REGION Network 7: 380A1 FB
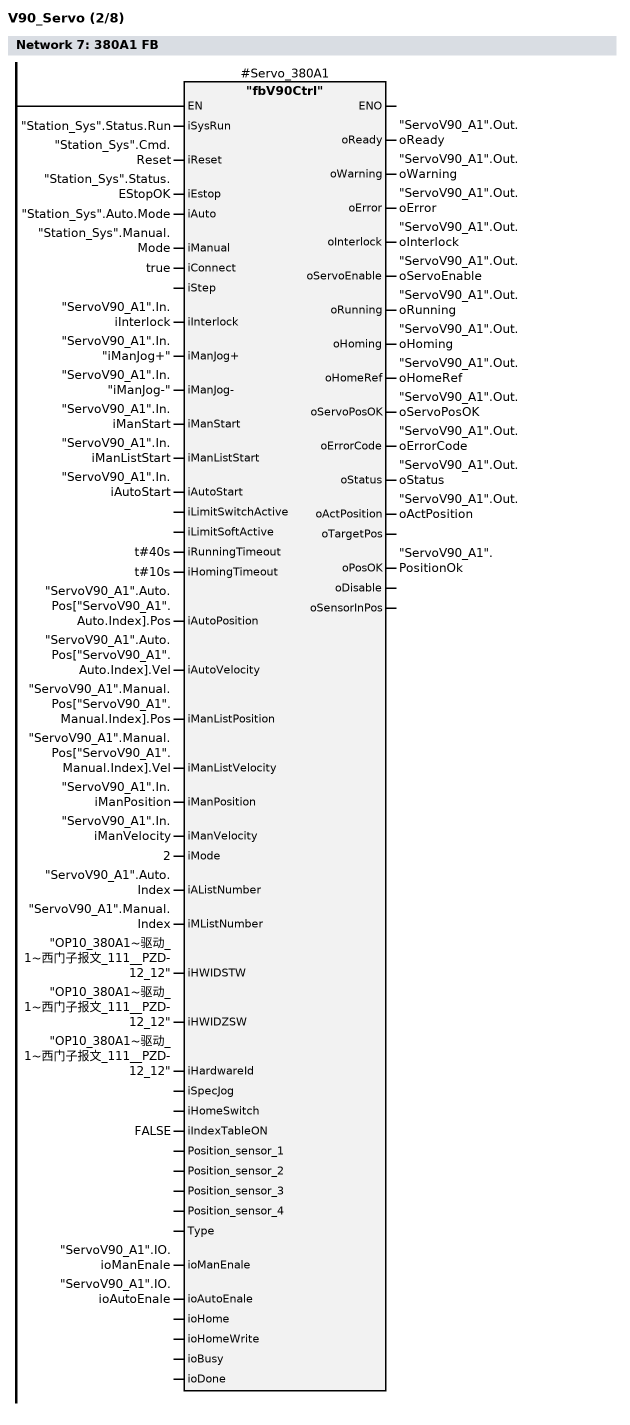
   RUNG wire#powerrail
      #Servo_380A1(iSysRun := "Station_Sys".Status.Run, iReset := "Station_Sys".Cmd.Reset, iEstop := "Station_Sys".Status.EStopOK, iAuto := "Station_Sys".Auto.Mode, iManual := "Station_Sys".Manual.Mode, iConnect := true, iStep :=, iInterlock := "ServoV90_A1".In.iInterlock, "iManJog+" := "ServoV90_A1".In."iManJog+", "iManJog-" := "ServoV90_A1".In."iManJog-", iManStart := "ServoV90_A1".In.iManStart, iManListStart := "ServoV90_A1".In.iManListStart, iAutoStart := "ServoV90_A1".In.iAutoStart, iLimitSwitchActive :=, iLimitSoftActive :=, iRunningTimeout := t#40s, iHomingTimeout := t#10s, iAutoPosition := "ServoV90_A1".Auto.Pos["ServoV90_A1".Auto.Index].Pos, iAutoVelocity := "ServoV90_A1".Auto.Pos["ServoV90_A1".Auto.Index].Vel, iManListPosition := "ServoV90_A1".Manual.Pos["ServoV90_A1".Manual.Index].Pos, iManListVelocity := "ServoV90_A1".Manual.Pos["ServoV90_A1".Manual.Index].Vel, iManPosition := "ServoV90_A1".In.iManPosition, iManVelocity := "ServoV90_A1".In.iManVelocity, iMode := 2, iAListNumber := "ServoV90_A1".Auto.Index, iMListNumber := "ServoV90_A1".Manual.Index, iHWIDSTW := "OP10_380A1~驱动_1~西门子报文_111__PZD-12_12", iHWIDZSW := "OP10_380A1~驱动_1~西门子报文_111__PZD-12_12", iHardwareId := "OP10_380A1~驱动_1~西门子报文_111__PZD-12_12", iSpecJog :=, iHomeSwitch :=, iIndexTableON := FALSE, Position_sensor_1 :=, Position_sensor_2 :=, Position_sensor_3 :=, Position_sensor_4 :=, "Type" :=, ioManEnale := "ServoV90_A1".IO.ioManEnale, ioAutoEnale := "ServoV90_A1".IO.ioAutoEnale, ioHome :=, ioHomeWrite :=, ioBusy :=, ioDone :=, oReady => "ServoV90_A1".Out.oReady, oWarning => "ServoV90_A1".Out.oWarning, oError => "ServoV90_A1".Out.oError, oInterlock => "ServoV90_A1".Out.oInterlock, oServoEnable => "ServoV90_A1".Out.oServoEnable, oRunning => "ServoV90_A1".Out.oRunning, oHoming => "ServoV90_A1".Out.oHoming, oHomeRef => "ServoV90_A1".Out.oHomeRef, oServoPosOK => "ServoV90_A1".Out.oServoPosOK, oErrorCode => "ServoV90_A1".Out.oErrorCode, oStatus => "ServoV90_A1".Out.oStatus, oActPosition => "ServoV90_A1".Out.oActPosition, oTargetPos =>, oPosOK => "ServoV90_A1".PositionOk, oDisable =>, oSensorInPos =>)
   END_RUNG
   // the same network as SCL:
   #Servo_380A1(iSysRun := "Station_Sys".Status.Run,   // "fbV90Ctrl"
                iReset := "Station_Sys".Cmd.Reset,
                iEstop := "Station_Sys".Status.EStopOK,
                iAuto := "Station_Sys".Auto.Mode,
                iManual := "Station_Sys".Manual.Mode,
                iConnect := true,
                iInterlock := "ServoV90_A1".In.iInterlock,
                "iManJog+" := "ServoV90_A1".In."iManJog+",
                "iManJog-" := "ServoV90_A1".In."iManJog-",
                iManStart := "ServoV90_A1".In.iManStart,
                iManListStart := "ServoV90_A1".In.iManListStart,
                iAutoStart := "ServoV90_A1".In.iAutoStart,
                iRunningTimeout := t#40s,
                iHomingTimeout := t#10s,
                iAutoPosition := "ServoV90_A1".Auto.Pos["ServoV90_A1".Auto.Index].Pos,
                iAutoVelocity := "ServoV90_A1".Auto.Pos["ServoV90_A1".Auto.Index].Vel,
                iManListPosition := "ServoV90_A1".Manual.Pos["ServoV90_A1".Manual.Index].Pos,
                iManListVelocity := "ServoV90_A1".Manual.Pos["ServoV90_A1".Manual.Index].Vel,
                iManPosition := "ServoV90_A1".In.iManPosition,
                iManVelocity := "ServoV90_A1".In.iManVelocity,
                iMode := 2,
                iAListNumber := "ServoV90_A1".Auto.Index,
                iMListNumber := "ServoV90_A1".Manual.Index,
                iHWIDSTW := "OP10_380A1~驱动_1~西门子报文_111__PZD-12_12",
                iHWIDZSW := "OP10_380A1~驱动_1~西门子报文_111__PZD-12_12",
                iHardwareId := "OP10_380A1~驱动_1~西门子报文_111__PZD-12_12",
                iIndexTableON := FALSE,
                ioManEnale := "ServoV90_A1".IO.ioManEnale,
                ioAutoEnale := "ServoV90_A1".IO.ioAutoEnale,
                oReady => "ServoV90_A1".Out.oReady,
                oWarning => "ServoV90_A1".Out.oWarning,
                oError => "ServoV90_A1".Out.oError,
                oInterlock => "ServoV90_A1".Out.oInterlock,
                oServoEnable => "ServoV90_A1".Out.oServoEnable,
                oRunning => "ServoV90_A1".Out.oRunning,
                oHoming => "ServoV90_A1".Out.oHoming,
                oHomeRef => "ServoV90_A1".Out.oHomeRef,
                oServoPosOK => "ServoV90_A1".Out.oServoPosOK,
                oErrorCode => "ServoV90_A1".Out.oErrorCode,
                oStatus => "ServoV90_A1".Out.oStatus,
                oActPosition => "ServoV90_A1".Out.oActPosition,
                oPosOK => "ServoV90_A1".PositionOk);
END_REGION

REGION Network 8 (SCL): 故障显示 / Fault indication
   //"ST70_DeviceError".Servo1.ServoDriverError := "ServoV90_A1".Out.oError;
END_REGION

REGION Network 9: <<<<<<<<<<<<<<<<<<<<<381A1 Servo>>>>>>>>>>>>>>>>>>>>>>>>>
END_REGION

REGION Network 10: negtive motion/action/...automaticly
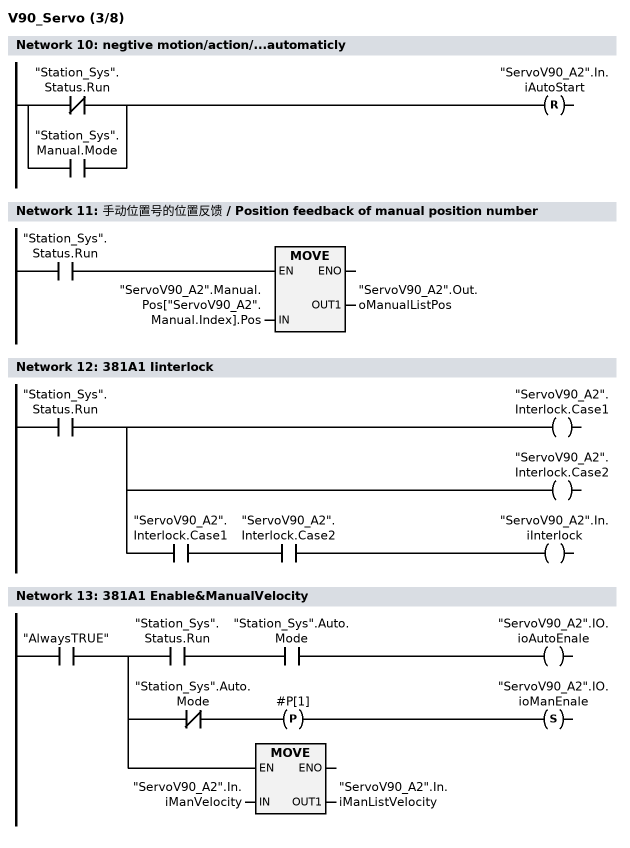
   RUNG wire#powerrail
      I_Contact( "Station_Sys".Status.Run )
      wire#w1
      R_Coil( "ServoV90_A2".In.iAutoStart )
   END_RUNG
   RUNG wire#powerrail
      Contact( "Station_Sys".Manual.Mode )
   END_RUNG wire#w1
   // the same network as SCL:
   IF NOT "Station_Sys".Status.Run OR "Station_Sys".Manual.Mode THEN
       "ServoV90_A2".In.iAutoStart := FALSE;
   END_IF;
END_REGION

REGION Network 11: 手动位置号的位置反馈 / Position feedback of manual position number
   RUNG wire#powerrail
      Contact( "Station_Sys".Status.Run )
      Move(in := "ServoV90_A2".Manual.Pos["ServoV90_A2".Manual.Index].Pos, out1 => "ServoV90_A2".Out.oManualListPos)
   END_RUNG
   // the same network as SCL:
   IF "Station_Sys".Status.Run THEN
       "ServoV90_A2".Out.oManualListPos := "ServoV90_A2".Manual.Pos["ServoV90_A2".Manual.Index].Pos;
   END_IF;
END_REGION

REGION Network 12: 381A1 Iinterlock
   RUNG wire#powerrail
      Contact( "Station_Sys".Status.Run )
      wire#w1
      Coil( "ServoV90_A2".Interlock.Case1 )
   END_RUNG
   RUNG wire#w1
      Coil( "ServoV90_A2".Interlock.Case2 )
   END_RUNG
   RUNG wire#w1
      Contact( "ServoV90_A2".Interlock.Case1 )
      Contact( "ServoV90_A2".Interlock.Case2 )
      Coil( "ServoV90_A2".In.iInterlock )
   END_RUNG
   // the same network as SCL:
   "ServoV90_A2".Interlock.Case1 := "Station_Sys".Status.Run;
   "ServoV90_A2".Interlock.Case2 := "Station_Sys".Status.Run;
   "ServoV90_A2".In.iInterlock := "Station_Sys".Status.Run AND "ServoV90_A2".Interlock.Case1 AND "ServoV90_A2".Interlock.Case2;
END_REGION

REGION Network 13: 381A1 Enable&ManualVelocity
   RUNG wire#powerrail
      Contact( "AlwaysTRUE" )
      wire#w1
      Contact( "Station_Sys".Status.Run )
      Contact( "Station_Sys".Auto.Mode )
      Coil( "ServoV90_A2".IO.ioAutoEnale )
   END_RUNG
   RUNG wire#w1
      I_Contact( "Station_Sys".Auto.Mode )
      P_Trig( #P[1] )
      S_Coil( "ServoV90_A2".IO.ioManEnale )
   END_RUNG
   RUNG wire#w1
      Move(in := "ServoV90_A2".In.iManVelocity, out1 => "ServoV90_A2".In.iManListVelocity)
   END_RUNG
   // the same network as SCL:
   "ServoV90_A2".IO.ioAutoEnale := "AlwaysTRUE" AND "Station_Sys".Status.Run AND "Station_Sys".Auto.Mode;
   #_w1 := "AlwaysTRUE" AND NOT "Station_Sys".Auto.Mode;
   #_w2 := #_w1 AND NOT #P[1];   // rising edge
   #P[1] := #_w1;
   IF #_w2 THEN "ServoV90_A2".IO.ioManEnale := TRUE; END_IF;
   IF "AlwaysTRUE" THEN "ServoV90_A2".In.iManListVelocity := "ServoV90_A2".In.iManVelocity; END_IF;
END_REGION

REGION Network 14 (SCL): 381A1 RecipePosition
    IF "Station_Sys".Status.Run THEN
        "ServoV90_A2".Manual.Pos[1].Pos := "ServoV90_A2".Auto.Pos[1].Pos := REAL_TO_DINT("Parameter".AxisRun.Axis[2].Pos1.Position*1000);
       "ServoV90_A2".Manual.Pos[1].Vel := "ServoV90_A2".Auto.Pos[1].Vel := "Parameter".AxisRun.Axis[2].Pos1.Speed;

       "ServoV90_A2".Manual.Pos[2].Pos := "ServoV90_A2".Auto.Pos[2].Pos := REAL_TO_DINT("Parameter".AxisRun.Axis[2].Pos2.Position*1000);
       "ServoV90_A2".Manual.Pos[2].Vel := "ServoV90_A2".Auto.Pos[2].Vel := "Parameter".AxisRun.Axis[2].Pos2.Speed;

       "ServoV90_A2".Manual.Pos[3].Pos := "ServoV90_A2".Auto.Pos[3].Pos := REAL_TO_DINT("Parameter".AxisRun.Axis[2].Pos3.Position*1000);
       "ServoV90_A2".Manual.Pos[3].Vel := "ServoV90_A2".Auto.Pos[3].Vel := "Parameter".AxisRun.Axis[2].Pos3.Speed;

       "ServoV90_A2".Manual.Pos[4].Pos := "ServoV90_A2".Auto.Pos[4].Pos := REAL_TO_DINT("Parameter".AxisRun.Axis[2].Pos4.Position*1000);
       "ServoV90_A2".Manual.Pos[4].Vel := "ServoV90_A2".Auto.Pos[4].Vel := "Parameter".AxisRun.Axis[2].Pos4.Speed;

       "ServoV90_A2".Manual.Pos[5].Pos := "ServoV90_A2".Auto.Pos[5].Pos := REAL_TO_DINT("Parameter".AxisRun.Axis[2].Pos5.Position*1000);
       "ServoV90_A2".Manual.Pos[5].Vel := "ServoV90_A2".Auto.Pos[5].Vel := "Parameter".AxisRun.Axis[2].Pos5.Speed;

       "ServoV90_A2".Manual.Pos[6].Pos := "ServoV90_A2".Auto.Pos[6].Pos := REAL_TO_DINT("Parameter".AxisRun.Axis[2].Pos6.Position*1000);
       "ServoV90_A2".Manual.Pos[6].Vel := "ServoV90_A2".Auto.Pos[6].Vel := "Parameter".AxisRun.Axis[2].Pos6.Speed;

       "ServoV90_A2".Manual.Pos[7].Pos := "ServoV90_A2".Auto.Pos[7].Pos := REAL_TO_DINT("Parameter".AxisRun.Axis[2].Pos7.Position*1000);
       "ServoV90_A2".Manual.Pos[7].Vel := "ServoV90_A2".Auto.Pos[7].Vel := "Parameter".AxisRun.Axis[2].Pos7.Speed;

       "ServoV90_A2".Manual.Pos[8].Pos := "ServoV90_A2".Auto.Pos[8].Pos := REAL_TO_DINT("Parameter".AxisRun.Axis[2].Pos8.Position*1000);
       "ServoV90_A2".Manual.Pos[8].Vel := "ServoV90_A2".Auto.Pos[8].Vel := "Parameter".AxisRun.Axis[2].Pos8.Speed;

       "ServoV90_A2".Manual.Pos[9].Pos := "ServoV90_A2".Auto.Pos[9].Pos := REAL_TO_DINT("Parameter".AxisRun.Axis[2].Pos9.Position*1000);
       "ServoV90_A2".Manual.Pos[9].Vel := "ServoV90_A2".Auto.Pos[9].Vel := "Parameter".AxisRun.Axis[2].Pos9.Speed;

       "ServoV90_A2".Manual.Pos[10].Pos := "ServoV90_A2".Auto.Pos[10].Pos := REAL_TO_DINT("Parameter".AxisRun.Axis[2].Pos10.Position*1000);
       "ServoV90_A2".Manual.Pos[10].Vel := "ServoV90_A2".Auto.Pos[10].Vel := "Parameter".AxisRun.Axis[2].Pos10.Speed;
   END_IF;
END_REGION

REGION Network 15: 381A1 FB
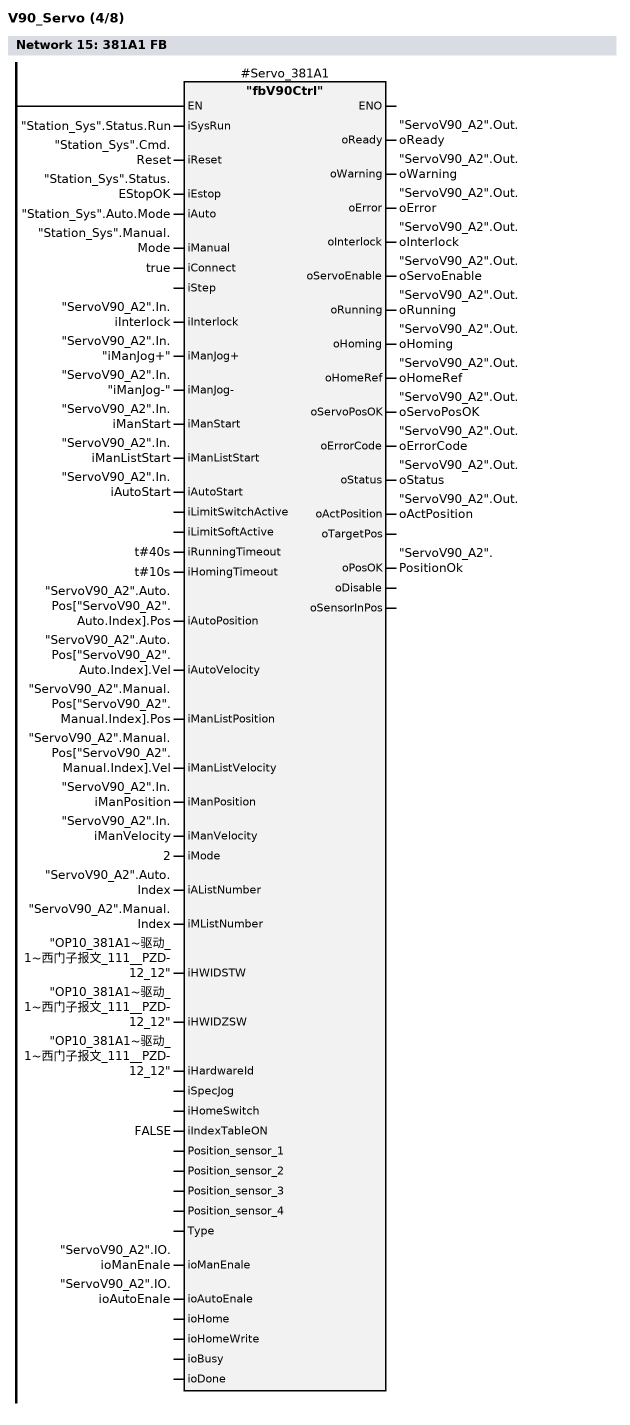
   RUNG wire#powerrail
      #Servo_381A1(iSysRun := "Station_Sys".Status.Run, iReset := "Station_Sys".Cmd.Reset, iEstop := "Station_Sys".Status.EStopOK, iAuto := "Station_Sys".Auto.Mode, iManual := "Station_Sys".Manual.Mode, iConnect := true, iStep :=, iInterlock := "ServoV90_A2".In.iInterlock, "iManJog+" := "ServoV90_A2".In."iManJog+", "iManJog-" := "ServoV90_A2".In."iManJog-", iManStart := "ServoV90_A2".In.iManStart, iManListStart := "ServoV90_A2".In.iManListStart, iAutoStart := "ServoV90_A2".In.iAutoStart, iLimitSwitchActive :=, iLimitSoftActive :=, iRunningTimeout := t#40s, iHomingTimeout := t#10s, iAutoPosition := "ServoV90_A2".Auto.Pos["ServoV90_A2".Auto.Index].Pos, iAutoVelocity := "ServoV90_A2".Auto.Pos["ServoV90_A2".Auto.Index].Vel, iManListPosition := "ServoV90_A2".Manual.Pos["ServoV90_A2".Manual.Index].Pos, iManListVelocity := "ServoV90_A2".Manual.Pos["ServoV90_A2".Manual.Index].Vel, iManPosition := "ServoV90_A2".In.iManPosition, iManVelocity := "ServoV90_A2".In.iManVelocity, iMode := 2, iAListNumber := "ServoV90_A2".Auto.Index, iMListNumber := "ServoV90_A2".Manual.Index, iHWIDSTW := "OP10_381A1~驱动_1~西门子报文_111__PZD-12_12", iHWIDZSW := "OP10_381A1~驱动_1~西门子报文_111__PZD-12_12", iHardwareId := "OP10_381A1~驱动_1~西门子报文_111__PZD-12_12", iSpecJog :=, iHomeSwitch :=, iIndexTableON := FALSE, Position_sensor_1 :=, Position_sensor_2 :=, Position_sensor_3 :=, Position_sensor_4 :=, "Type" :=, ioManEnale := "ServoV90_A2".IO.ioManEnale, ioAutoEnale := "ServoV90_A2".IO.ioAutoEnale, ioHome :=, ioHomeWrite :=, ioBusy :=, ioDone :=, oReady => "ServoV90_A2".Out.oReady, oWarning => "ServoV90_A2".Out.oWarning, oError => "ServoV90_A2".Out.oError, oInterlock => "ServoV90_A2".Out.oInterlock, oServoEnable => "ServoV90_A2".Out.oServoEnable, oRunning => "ServoV90_A2".Out.oRunning, oHoming => "ServoV90_A2".Out.oHoming, oHomeRef => "ServoV90_A2".Out.oHomeRef, oServoPosOK => "ServoV90_A2".Out.oServoPosOK, oErrorCode => "ServoV90_A2".Out.oErrorCode, oStatus => "ServoV90_A2".Out.oStatus, oActPosition => "ServoV90_A2".Out.oActPosition, oTargetPos =>, oPosOK => "ServoV90_A2".PositionOk, oDisable =>, oSensorInPos =>)
   END_RUNG
   // the same network as SCL:
   #Servo_381A1(iSysRun := "Station_Sys".Status.Run,   // "fbV90Ctrl"
                iReset := "Station_Sys".Cmd.Reset,
                iEstop := "Station_Sys".Status.EStopOK,
                iAuto := "Station_Sys".Auto.Mode,
                iManual := "Station_Sys".Manual.Mode,
                iConnect := true,
                iInterlock := "ServoV90_A2".In.iInterlock,
                "iManJog+" := "ServoV90_A2".In."iManJog+",
                "iManJog-" := "ServoV90_A2".In."iManJog-",
                iManStart := "ServoV90_A2".In.iManStart,
                iManListStart := "ServoV90_A2".In.iManListStart,
                iAutoStart := "ServoV90_A2".In.iAutoStart,
                iRunningTimeout := t#40s,
                iHomingTimeout := t#10s,
                iAutoPosition := "ServoV90_A2".Auto.Pos["ServoV90_A2".Auto.Index].Pos,
                iAutoVelocity := "ServoV90_A2".Auto.Pos["ServoV90_A2".Auto.Index].Vel,
                iManListPosition := "ServoV90_A2".Manual.Pos["ServoV90_A2".Manual.Index].Pos,
                iManListVelocity := "ServoV90_A2".Manual.Pos["ServoV90_A2".Manual.Index].Vel,
                iManPosition := "ServoV90_A2".In.iManPosition,
                iManVelocity := "ServoV90_A2".In.iManVelocity,
                iMode := 2,
                iAListNumber := "ServoV90_A2".Auto.Index,
                iMListNumber := "ServoV90_A2".Manual.Index,
                iHWIDSTW := "OP10_381A1~驱动_1~西门子报文_111__PZD-12_12",
                iHWIDZSW := "OP10_381A1~驱动_1~西门子报文_111__PZD-12_12",
                iHardwareId := "OP10_381A1~驱动_1~西门子报文_111__PZD-12_12",
                iIndexTableON := FALSE,
                ioManEnale := "ServoV90_A2".IO.ioManEnale,
                ioAutoEnale := "ServoV90_A2".IO.ioAutoEnale,
                oReady => "ServoV90_A2".Out.oReady,
                oWarning => "ServoV90_A2".Out.oWarning,
                oError => "ServoV90_A2".Out.oError,
                oInterlock => "ServoV90_A2".Out.oInterlock,
                oServoEnable => "ServoV90_A2".Out.oServoEnable,
                oRunning => "ServoV90_A2".Out.oRunning,
                oHoming => "ServoV90_A2".Out.oHoming,
                oHomeRef => "ServoV90_A2".Out.oHomeRef,
                oServoPosOK => "ServoV90_A2".Out.oServoPosOK,
                oErrorCode => "ServoV90_A2".Out.oErrorCode,
                oStatus => "ServoV90_A2".Out.oStatus,
                oActPosition => "ServoV90_A2".Out.oActPosition,
                oPosOK => "ServoV90_A2".PositionOk);
END_REGION

REGION Network 16 (SCL): 故障显示 / Fault indication
   //"ST70_DeviceError".Servo2.ServoDriverError := "ServoV90_A2".Out.oError;
END_REGION

REGION Network 17: <<<<<<<<<<<<<<<<<<<<<382A1 Servo>>>>>>>>>>>>>>>>>>>>>>>>>
END_REGION

REGION Network 18: negtive motion/action/...automaticly
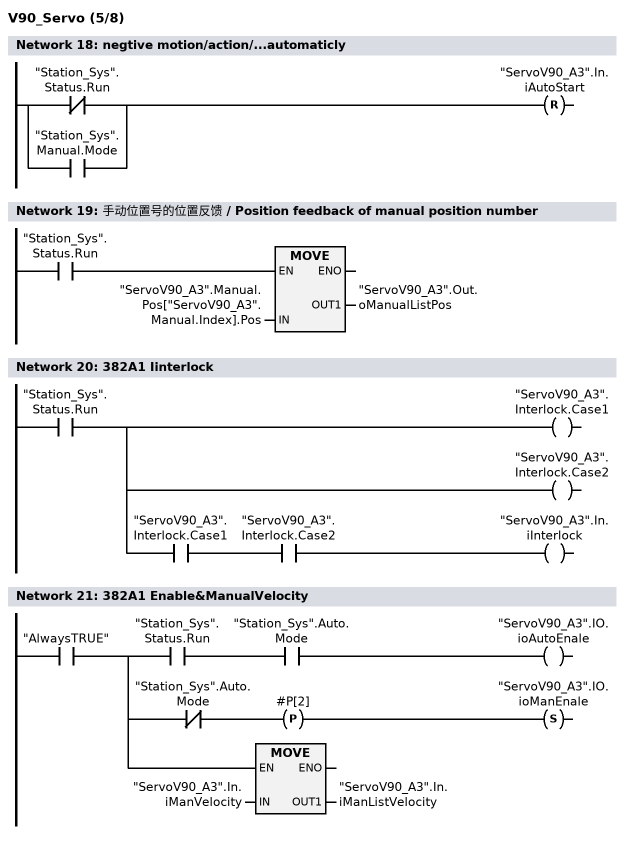
   RUNG wire#powerrail
      I_Contact( "Station_Sys".Status.Run )
      wire#w1
      R_Coil( "ServoV90_A3".In.iAutoStart )
   END_RUNG
   RUNG wire#powerrail
      Contact( "Station_Sys".Manual.Mode )
   END_RUNG wire#w1
   // the same network as SCL:
   IF NOT "Station_Sys".Status.Run OR "Station_Sys".Manual.Mode THEN
       "ServoV90_A3".In.iAutoStart := FALSE;
   END_IF;
END_REGION

REGION Network 19: 手动位置号的位置反馈 / Position feedback of manual position number
   RUNG wire#powerrail
      Contact( "Station_Sys".Status.Run )
      Move(in := "ServoV90_A3".Manual.Pos["ServoV90_A3".Manual.Index].Pos, out1 => "ServoV90_A3".Out.oManualListPos)
   END_RUNG
   // the same network as SCL:
   IF "Station_Sys".Status.Run THEN
       "ServoV90_A3".Out.oManualListPos := "ServoV90_A3".Manual.Pos["ServoV90_A3".Manual.Index].Pos;
   END_IF;
END_REGION

REGION Network 20: 382A1 Iinterlock
   RUNG wire#powerrail
      Contact( "Station_Sys".Status.Run )
      wire#w1
      Coil( "ServoV90_A3".Interlock.Case1 )
   END_RUNG
   RUNG wire#w1
      Coil( "ServoV90_A3".Interlock.Case2 )
   END_RUNG
   RUNG wire#w1
      Contact( "ServoV90_A3".Interlock.Case1 )
      Contact( "ServoV90_A3".Interlock.Case2 )
      Coil( "ServoV90_A3".In.iInterlock )
   END_RUNG
   // the same network as SCL:
   "ServoV90_A3".Interlock.Case1 := "Station_Sys".Status.Run;
   "ServoV90_A3".Interlock.Case2 := "Station_Sys".Status.Run;
   "ServoV90_A3".In.iInterlock := "Station_Sys".Status.Run AND "ServoV90_A3".Interlock.Case1 AND "ServoV90_A3".Interlock.Case2;
END_REGION

REGION Network 21: 382A1 Enable&ManualVelocity
   RUNG wire#powerrail
      Contact( "AlwaysTRUE" )
      wire#w1
      Contact( "Station_Sys".Status.Run )
      Contact( "Station_Sys".Auto.Mode )
      Coil( "ServoV90_A3".IO.ioAutoEnale )
   END_RUNG
   RUNG wire#w1
      I_Contact( "Station_Sys".Auto.Mode )
      P_Trig( #P[2] )
      S_Coil( "ServoV90_A3".IO.ioManEnale )
   END_RUNG
   RUNG wire#w1
      Move(in := "ServoV90_A3".In.iManVelocity, out1 => "ServoV90_A3".In.iManListVelocity)
   END_RUNG
   // the same network as SCL:
   "ServoV90_A3".IO.ioAutoEnale := "AlwaysTRUE" AND "Station_Sys".Status.Run AND "Station_Sys".Auto.Mode;
   #_w1 := "AlwaysTRUE" AND NOT "Station_Sys".Auto.Mode;
   #_w2 := #_w1 AND NOT #P[2];   // rising edge
   #P[2] := #_w1;
   IF #_w2 THEN "ServoV90_A3".IO.ioManEnale := TRUE; END_IF;
   IF "AlwaysTRUE" THEN "ServoV90_A3".In.iManListVelocity := "ServoV90_A3".In.iManVelocity; END_IF;
END_REGION

REGION Network 22 (SCL): 382A1 RecipePosition
    IF "Station_Sys".Status.Run THEN
        "ServoV90_A3".Manual.Pos[1].Pos := "ServoV90_A3".Auto.Pos[1].Pos := REAL_TO_DINT("Parameter".AxisRun.Axis[3].Pos1.Position*1000);
        "ServoV90_A3".Manual.Pos[1].Vel := "ServoV90_A3".Auto.Pos[1].Vel := "Parameter".AxisRun.Axis[3].Pos1.Speed;

        "ServoV90_A3".Manual.Pos[2].Pos := "ServoV90_A3".Auto.Pos[2].Pos := REAL_TO_DINT("Parameter".AxisRun.Axis[3].Pos2.Position*1000);
        "ServoV90_A3".Manual.Pos[2].Vel := "ServoV90_A3".Auto.Pos[2].Vel := "Parameter".AxisRun.Axis[3].Pos2.Speed;

        "ServoV90_A3".Manual.Pos[3].Pos := "ServoV90_A3".Auto.Pos[3].Pos := REAL_TO_DINT("Parameter".AxisRun.Axis[3].Pos3.Position*1000);
        "ServoV90_A3".Manual.Pos[3].Vel := "ServoV90_A3".Auto.Pos[3].Vel := "Parameter".AxisRun.Axis[3].Pos3.Speed;

        "ServoV90_A3".Manual.Pos[4].Pos := "ServoV90_A3".Auto.Pos[4].Pos := REAL_TO_DINT("Parameter".AxisRun.Axis[3].Pos4.Position*1000);
        "ServoV90_A3".Manual.Pos[4].Vel := "ServoV90_A3".Auto.Pos[4].Vel := "Parameter".AxisRun.Axis[3].Pos4.Speed;

        "ServoV90_A3".Manual.Pos[5].Pos := "ServoV90_A3".Auto.Pos[5].Pos := REAL_TO_DINT("Parameter".AxisRun.Axis[3].Pos5.Position*1000);
        "ServoV90_A3".Manual.Pos[5].Vel := "ServoV90_A3".Auto.Pos[5].Vel := "Parameter".AxisRun.Axis[3].Pos5.Speed;

        "ServoV90_A3".Manual.Pos[6].Pos := "ServoV90_A3".Auto.Pos[6].Pos := REAL_TO_DINT("Parameter".AxisRun.Axis[3].Pos6.Position*1000);
        "ServoV90_A3".Manual.Pos[6].Vel := "ServoV90_A3".Auto.Pos[6].Vel := "Parameter".AxisRun.Axis[3].Pos6.Speed;

        "ServoV90_A3".Manual.Pos[7].Pos := "ServoV90_A3".Auto.Pos[7].Pos := REAL_TO_DINT("Parameter".AxisRun.Axis[3].Pos7.Position*1000);
        "ServoV90_A3".Manual.Pos[7].Vel := "ServoV90_A3".Auto.Pos[7].Vel := "Parameter".AxisRun.Axis[3].Pos7.Speed;

        "ServoV90_A3".Manual.Pos[8].Pos := "ServoV90_A3".Auto.Pos[8].Pos := REAL_TO_DINT("Parameter".AxisRun.Axis[3].Pos8.Position*1000);
        "ServoV90_A3".Manual.Pos[8].Vel := "ServoV90_A3".Auto.Pos[8].Vel := "Parameter".AxisRun.Axis[3].Pos8.Speed;

        "ServoV90_A3".Manual.Pos[9].Pos := "ServoV90_A3".Auto.Pos[9].Pos := REAL_TO_DINT("Parameter".AxisRun.Axis[3].Pos9.Position*1000);
        "ServoV90_A3".Manual.Pos[9].Vel := "ServoV90_A3".Auto.Pos[9].Vel := "Parameter".AxisRun.Axis[3].Pos9.Speed;

        "ServoV90_A3".Manual.Pos[10].Pos := "ServoV90_A3".Auto.Pos[10].Pos := REAL_TO_DINT("Parameter".AxisRun.Axis[3].Pos10.Position*1000);
        "ServoV90_A3".Manual.Pos[10].Vel := "ServoV90_A3".Auto.Pos[10].Vel := "Parameter".AxisRun.Axis[3].Pos10.Speed;
   END_IF;
END_REGION

REGION Network 23: 382A1 FB
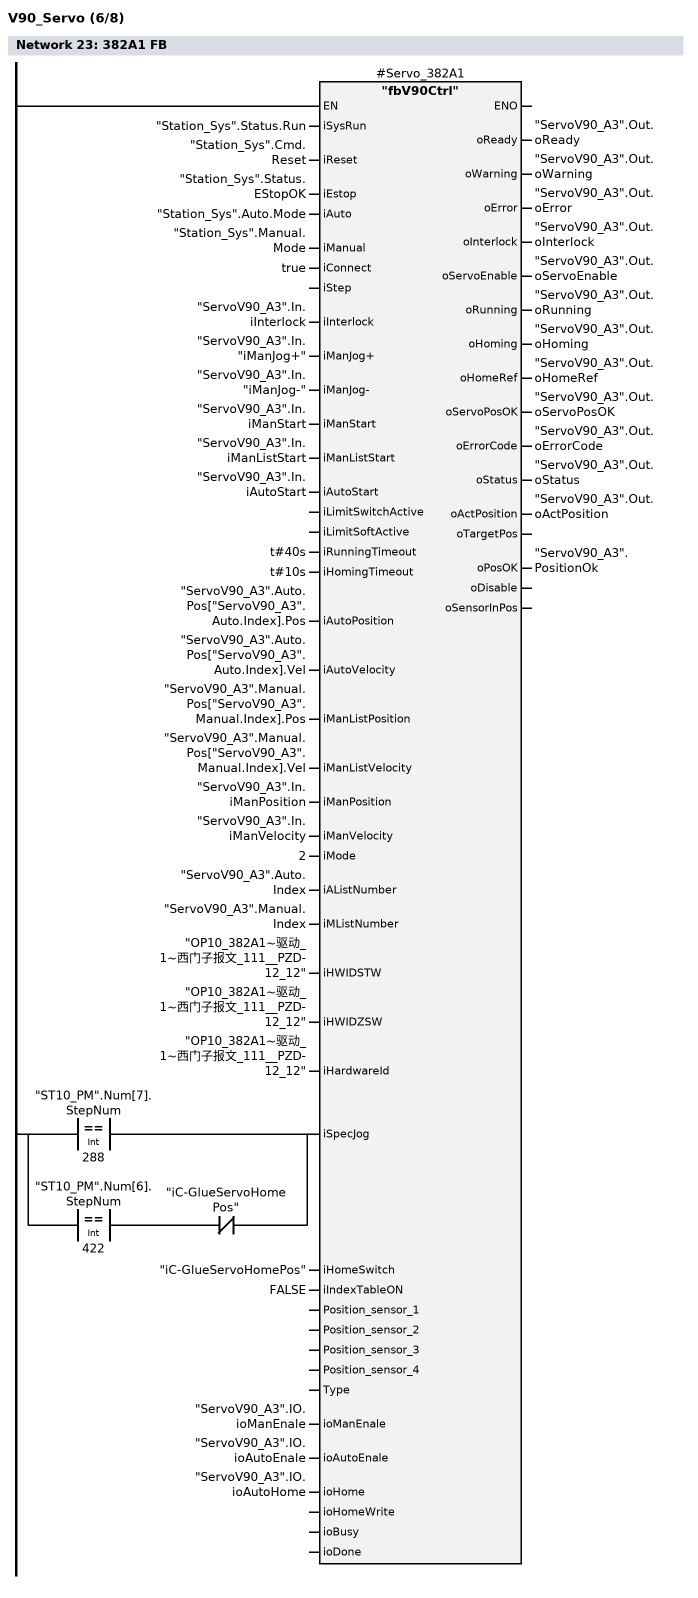
   RUNG wire#powerrail
      #Servo_382A1(iSpecJog := wire#w1, iSysRun := "Station_Sys".Status.Run, iReset := "Station_Sys".Cmd.Reset, iEstop := "Station_Sys".Status.EStopOK, iAuto := "Station_Sys".Auto.Mode, iManual := "Station_Sys".Manual.Mode, iConnect := true, iStep :=, iInterlock := "ServoV90_A3".In.iInterlock, "iManJog+" := "ServoV90_A3".In."iManJog+", "iManJog-" := "ServoV90_A3".In."iManJog-", iManStart := "ServoV90_A3".In.iManStart, iManListStart := "ServoV90_A3".In.iManListStart, iAutoStart := "ServoV90_A3".In.iAutoStart, iLimitSwitchActive :=, iLimitSoftActive :=, iRunningTimeout := t#40s, iHomingTimeout := t#10s, iAutoPosition := "ServoV90_A3".Auto.Pos["ServoV90_A3".Auto.Index].Pos, iAutoVelocity := "ServoV90_A3".Auto.Pos["ServoV90_A3".Auto.Index].Vel, iManListPosition := "ServoV90_A3".Manual.Pos["ServoV90_A3".Manual.Index].Pos, iManListVelocity := "ServoV90_A3".Manual.Pos["ServoV90_A3".Manual.Index].Vel, iManPosition := "ServoV90_A3".In.iManPosition, iManVelocity := "ServoV90_A3".In.iManVelocity, iMode := 2, iAListNumber := "ServoV90_A3".Auto.Index, iMListNumber := "ServoV90_A3".Manual.Index, iHWIDSTW := "OP10_382A1~驱动_1~西门子报文_111__PZD-12_12", iHWIDZSW := "OP10_382A1~驱动_1~西门子报文_111__PZD-12_12", iHardwareId := "OP10_382A1~驱动_1~西门子报文_111__PZD-12_12", iHomeSwitch := "iC-GlueServoHomePos", iIndexTableON := FALSE, Position_sensor_1 :=, Position_sensor_2 :=, Position_sensor_3 :=, Position_sensor_4 :=, "Type" :=, ioManEnale := "ServoV90_A3".IO.ioManEnale, ioAutoEnale := "ServoV90_A3".IO.ioAutoEnale, ioHome := "ServoV90_A3".IO.ioAutoHome, ioHomeWrite :=, ioBusy :=, ioDone :=, oReady => "ServoV90_A3".Out.oReady, oWarning => "ServoV90_A3".Out.oWarning, oError => "ServoV90_A3".Out.oError, oInterlock => "ServoV90_A3".Out.oInterlock, oServoEnable => "ServoV90_A3".Out.oServoEnable, oRunning => "ServoV90_A3".Out.oRunning, oHoming => "ServoV90_A3".Out.oHoming, oHomeRef => "ServoV90_A3".Out.oHomeRef, oServoPosOK => "ServoV90_A3".Out.oServoPosOK, oErrorCode => "ServoV90_A3".Out.oErrorCode, oStatus => "ServoV90_A3".Out.oStatus, oActPosition => "ServoV90_A3".Out.oActPosition, oTargetPos =>, oPosOK => "ServoV90_A3".PositionOk, oDisable =>, oSensorInPos =>)
   END_RUNG
   RUNG wire#powerrail
      { S7_Templates := "SrcType := Int" } EQ_Contact(in1 := "ST10_PM".Num[7].StepNum, in2 := 288)
   END_RUNG wire#w1
   RUNG wire#powerrail
      { S7_Templates := "SrcType := Int" } EQ_Contact(in1 := "ST10_PM".Num[6].StepNum, in2 := 422)
      I_Contact( "iC-GlueServoHomePos" )
   END_RUNG wire#w1
   // the same network as SCL:
   #Servo_382A1(iSysRun := "Station_Sys".Status.Run,   // "fbV90Ctrl"
                iReset := "Station_Sys".Cmd.Reset,
                iEstop := "Station_Sys".Status.EStopOK,
                iAuto := "Station_Sys".Auto.Mode,
                iManual := "Station_Sys".Manual.Mode,
                iConnect := true,
                iInterlock := "ServoV90_A3".In.iInterlock,
                "iManJog+" := "ServoV90_A3".In."iManJog+",
                "iManJog-" := "ServoV90_A3".In."iManJog-",
                iManStart := "ServoV90_A3".In.iManStart,
                iManListStart := "ServoV90_A3".In.iManListStart,
                iAutoStart := "ServoV90_A3".In.iAutoStart,
                iRunningTimeout := t#40s,
                iHomingTimeout := t#10s,
                iAutoPosition := "ServoV90_A3".Auto.Pos["ServoV90_A3".Auto.Index].Pos,
                iAutoVelocity := "ServoV90_A3".Auto.Pos["ServoV90_A3".Auto.Index].Vel,
                iManListPosition := "ServoV90_A3".Manual.Pos["ServoV90_A3".Manual.Index].Pos,
                iManListVelocity := "ServoV90_A3".Manual.Pos["ServoV90_A3".Manual.Index].Vel,
                iManPosition := "ServoV90_A3".In.iManPosition,
                iManVelocity := "ServoV90_A3".In.iManVelocity,
                iMode := 2,
                iAListNumber := "ServoV90_A3".Auto.Index,
                iMListNumber := "ServoV90_A3".Manual.Index,
                iHWIDSTW := "OP10_382A1~驱动_1~西门子报文_111__PZD-12_12",
                iHWIDZSW := "OP10_382A1~驱动_1~西门子报文_111__PZD-12_12",
                iHardwareId := "OP10_382A1~驱动_1~西门子报文_111__PZD-12_12",
                iSpecJog := ("ST10_PM".Num[7].StepNum = 288) OR (("ST10_PM".Num[6].StepNum = 422) AND NOT "iC-GlueServoHomePos"),
                iHomeSwitch := "iC-GlueServoHomePos",
                iIndexTableON := FALSE,
                ioManEnale := "ServoV90_A3".IO.ioManEnale,
                ioAutoEnale := "ServoV90_A3".IO.ioAutoEnale,
                ioHome := "ServoV90_A3".IO.ioAutoHome,
                oReady => "ServoV90_A3".Out.oReady,
                oWarning => "ServoV90_A3".Out.oWarning,
                oError => "ServoV90_A3".Out.oError,
                oInterlock => "ServoV90_A3".Out.oInterlock,
                oServoEnable => "ServoV90_A3".Out.oServoEnable,
                oRunning => "ServoV90_A3".Out.oRunning,
                oHoming => "ServoV90_A3".Out.oHoming,
                oHomeRef => "ServoV90_A3".Out.oHomeRef,
                oServoPosOK => "ServoV90_A3".Out.oServoPosOK,
                oErrorCode => "ServoV90_A3".Out.oErrorCode,
                oStatus => "ServoV90_A3".Out.oStatus,
                oActPosition => "ServoV90_A3".Out.oActPosition,
                oPosOK => "ServoV90_A3".PositionOk);
END_REGION

REGION Network 24: 复位启动
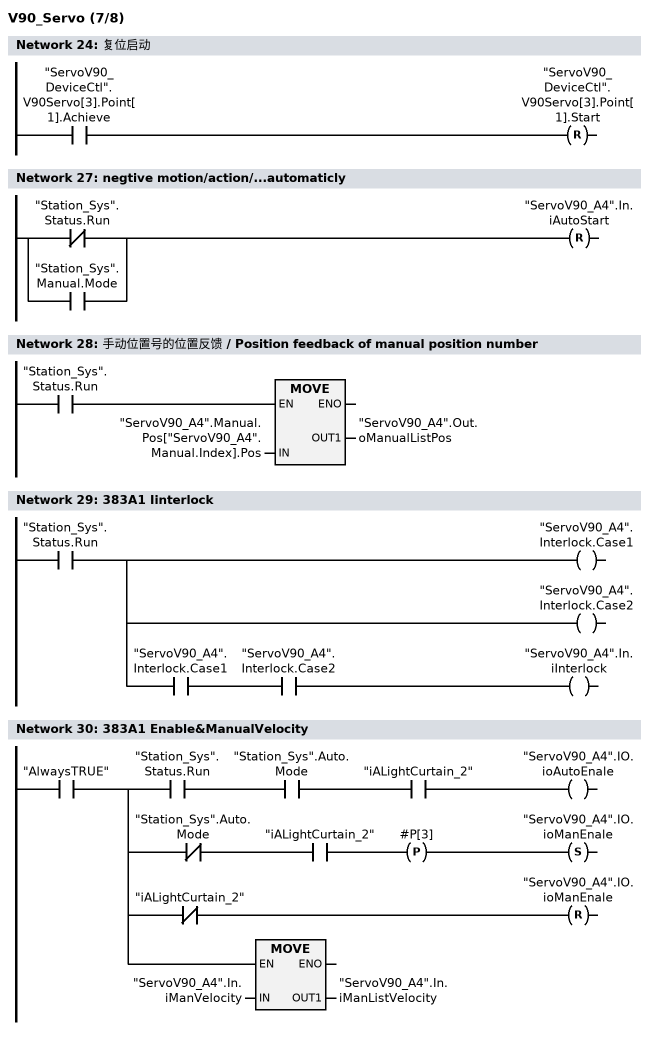
   RUNG wire#powerrail
      Contact( "ServoV90_DeviceCtl".V90Servo[3].Point[1].Achieve )
      R_Coil( "ServoV90_DeviceCtl".V90Servo[3].Point[1].Start )
   END_RUNG
   // the same network as SCL:
   IF "ServoV90_DeviceCtl".V90Servo[3].Point[1].Achieve THEN
       "ServoV90_DeviceCtl".V90Servo[3].Point[1].Start := FALSE;
   END_IF;
END_REGION

REGION Network 25 (SCL): 故障显示 / Fault indication
   //"ST70_DeviceError".Servo2.ServoDriverError := "ServoV90_A3".Out.oError;
END_REGION

REGION Network 26: <<<<<<<<<<<<<<<<<<<<<383A1 Servo>>>>>>>>>>>>>>>>>>>>>>>>>
END_REGION

REGION Network 27: negtive motion/action/...automaticly
   RUNG wire#powerrail
      I_Contact( "Station_Sys".Status.Run )
      wire#w1
      R_Coil( "ServoV90_A4".In.iAutoStart )
   END_RUNG
   RUNG wire#powerrail
      Contact( "Station_Sys".Manual.Mode )
   END_RUNG wire#w1
   // the same network as SCL:
   IF NOT "Station_Sys".Status.Run OR "Station_Sys".Manual.Mode THEN
       "ServoV90_A4".In.iAutoStart := FALSE;
   END_IF;
END_REGION

REGION Network 28: 手动位置号的位置反馈 / Position feedback of manual position number
   RUNG wire#powerrail
      Contact( "Station_Sys".Status.Run )
      Move(in := "ServoV90_A4".Manual.Pos["ServoV90_A4".Manual.Index].Pos, out1 => "ServoV90_A4".Out.oManualListPos)
   END_RUNG
   // the same network as SCL:
   IF "Station_Sys".Status.Run THEN
       "ServoV90_A4".Out.oManualListPos := "ServoV90_A4".Manual.Pos["ServoV90_A4".Manual.Index].Pos;
   END_IF;
END_REGION

REGION Network 29: 383A1 Iinterlock
   RUNG wire#powerrail
      Contact( "Station_Sys".Status.Run )
      wire#w1
      Coil( "ServoV90_A4".Interlock.Case1 )
   END_RUNG
   RUNG wire#w1
      Coil( "ServoV90_A4".Interlock.Case2 )
   END_RUNG
   RUNG wire#w1
      Contact( "ServoV90_A4".Interlock.Case1 )
      Contact( "ServoV90_A4".Interlock.Case2 )
      Coil( "ServoV90_A4".In.iInterlock )
   END_RUNG
   // the same network as SCL:
   "ServoV90_A4".Interlock.Case1 := "Station_Sys".Status.Run;
   "ServoV90_A4".Interlock.Case2 := "Station_Sys".Status.Run;
   "ServoV90_A4".In.iInterlock := "Station_Sys".Status.Run AND "ServoV90_A4".Interlock.Case1 AND "ServoV90_A4".Interlock.Case2;
END_REGION

REGION Network 30: 383A1 Enable&ManualVelocity
   RUNG wire#powerrail
      Contact( "AlwaysTRUE" )
      wire#w1
      Contact( "Station_Sys".Status.Run )
      Contact( "Station_Sys".Auto.Mode )
      Contact( "iALightCurtain_2" )
      Coil( "ServoV90_A4".IO.ioAutoEnale )
   END_RUNG
   RUNG wire#w1
      I_Contact( "Station_Sys".Auto.Mode )
      Contact( "iALightCurtain_2" )
      P_Trig( #P[3] )
      S_Coil( "ServoV90_A4".IO.ioManEnale )
   END_RUNG
   RUNG wire#w1
      I_Contact( "iALightCurtain_2" )
      R_Coil( "ServoV90_A4".IO.ioManEnale )
   END_RUNG
   RUNG wire#w1
      Move(in := "ServoV90_A4".In.iManVelocity, out1 => "ServoV90_A4".In.iManListVelocity)
   END_RUNG
   // the same network as SCL:
   "ServoV90_A4".IO.ioAutoEnale := "AlwaysTRUE" AND "Station_Sys".Status.Run AND "Station_Sys".Auto.Mode AND "iALightCurtain_2";
   #_w1 := "AlwaysTRUE" AND NOT "Station_Sys".Auto.Mode AND "iALightCurtain_2";
   #_w2 := #_w1 AND NOT #P[3];   // rising edge
   #P[3] := #_w1;
   IF #_w2 THEN "ServoV90_A4".IO.ioManEnale := TRUE; END_IF;
   IF "AlwaysTRUE" AND NOT "iALightCurtain_2" THEN "ServoV90_A4".IO.ioManEnale := FALSE; END_IF;
   IF "AlwaysTRUE" THEN "ServoV90_A4".In.iManListVelocity := "ServoV90_A4".In.iManVelocity; END_IF;
END_REGION

REGION Network 31 (SCL): 383A1 RecipePosition
   IF "Station_Sys".Status.Run THEN
       "ServoV90_A4".Manual.Pos[1].Pos := "ServoV90_A4".Auto.Pos[1].Pos := REAL_TO_DINT("Parameter".AxisRun.Axis[4].Pos1.Position*1000);
       "ServoV90_A4".Manual.Pos[1].Vel := "ServoV90_A4".Auto.Pos[1].Vel := "Parameter".AxisRun.Axis[4].Pos1.Speed;

       "ServoV90_A4".Manual.Pos[2].Pos := "ServoV90_A4".Auto.Pos[2].Pos := REAL_TO_DINT("Parameter".AxisRun.Axis[4].Pos2.Position*1000);
       "ServoV90_A4".Manual.Pos[2].Vel := "ServoV90_A4".Auto.Pos[2].Vel := "Parameter".AxisRun.Axis[4].Pos2.Speed;

       "ServoV90_A4".Manual.Pos[3].Pos := "ServoV90_A4".Auto.Pos[3].Pos := REAL_TO_DINT("Parameter".AxisRun.Axis[4].Pos3.Position*1000);
       "ServoV90_A4".Manual.Pos[3].Vel := "ServoV90_A4".Auto.Pos[3].Vel := "Parameter".AxisRun.Axis[4].Pos3.Speed;

       "ServoV90_A4".Manual.Pos[4].Pos := "ServoV90_A4".Auto.Pos[4].Pos := REAL_TO_DINT("Parameter".AxisRun.Axis[4].Pos4.Position*1000);
       "ServoV90_A4".Manual.Pos[4].Vel := "ServoV90_A4".Auto.Pos[4].Vel := "Parameter".AxisRun.Axis[4].Pos4.Speed;

       "ServoV90_A4".Manual.Pos[5].Pos := "ServoV90_A4".Auto.Pos[5].Pos := REAL_TO_DINT("Parameter".AxisRun.Axis[4].Pos5.Position*1000);
       "ServoV90_A4".Manual.Pos[5].Vel := "ServoV90_A4".Auto.Pos[5].Vel := "Parameter".AxisRun.Axis[4].Pos5.Speed;

       "ServoV90_A4".Manual.Pos[6].Pos := "ServoV90_A4".Auto.Pos[6].Pos := REAL_TO_DINT("Parameter".AxisRun.Axis[4].Pos6.Position*1000);
       "ServoV90_A4".Manual.Pos[6].Vel := "ServoV90_A4".Auto.Pos[6].Vel := "Parameter".AxisRun.Axis[4].Pos6.Speed;

       "ServoV90_A4".Manual.Pos[7].Pos := "ServoV90_A4".Auto.Pos[7].Pos := REAL_TO_DINT("Parameter".AxisRun.Axis[4].Pos7.Position*1000);
       "ServoV90_A4".Manual.Pos[7].Vel := "ServoV90_A4".Auto.Pos[7].Vel := "Parameter".AxisRun.Axis[4].Pos7.Speed;

       "ServoV90_A4".Manual.Pos[8].Pos := "ServoV90_A4".Auto.Pos[8].Pos := REAL_TO_DINT("Parameter".AxisRun.Axis[4].Pos8.Position*1000);
       "ServoV90_A4".Manual.Pos[8].Vel := "ServoV90_A4".Auto.Pos[8].Vel := "Parameter".AxisRun.Axis[4].Pos8.Speed;

       "ServoV90_A4".Manual.Pos[9].Pos := "ServoV90_A4".Auto.Pos[9].Pos := REAL_TO_DINT("Parameter".AxisRun.Axis[4].Pos9.Position*1000);
       "ServoV90_A4".Manual.Pos[9].Vel := "ServoV90_A4".Auto.Pos[9].Vel := "Parameter".AxisRun.Axis[4].Pos9.Speed;

       "ServoV90_A4".Manual.Pos[10].Pos := "ServoV90_A4".Auto.Pos[10].Pos := REAL_TO_DINT("Parameter".AxisRun.Axis[4].Pos10.Position*1000);
       "ServoV90_A4".Manual.Pos[10].Vel := "ServoV90_A4".Auto.Pos[10].Vel := "Parameter".AxisRun.Axis[4].Pos10.Speed;
   END_IF;
END_REGION

REGION Network 32: 383A1 FB
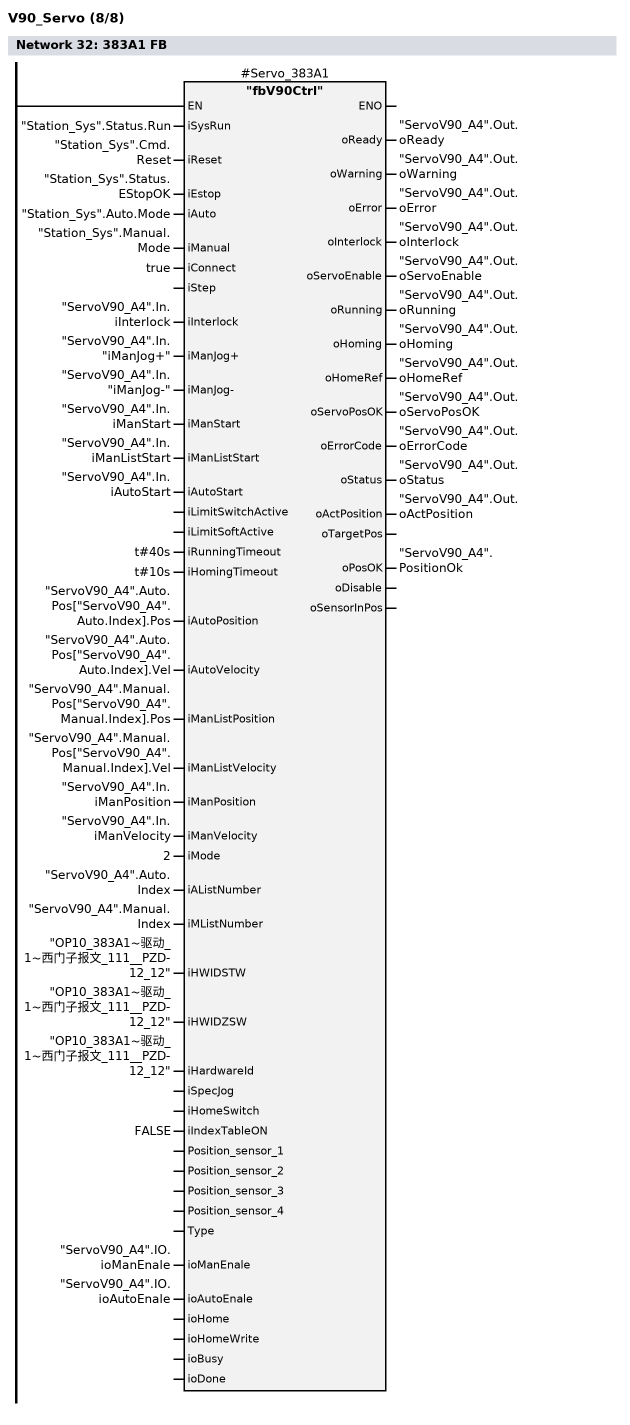
   RUNG wire#powerrail
      #Servo_383A1(iSysRun := "Station_Sys".Status.Run, iReset := "Station_Sys".Cmd.Reset, iEstop := "Station_Sys".Status.EStopOK, iAuto := "Station_Sys".Auto.Mode, iManual := "Station_Sys".Manual.Mode, iConnect := true, iStep :=, iInterlock := "ServoV90_A4".In.iInterlock, "iManJog+" := "ServoV90_A4".In."iManJog+", "iManJog-" := "ServoV90_A4".In."iManJog-", iManStart := "ServoV90_A4".In.iManStart, iManListStart := "ServoV90_A4".In.iManListStart, iAutoStart := "ServoV90_A4".In.iAutoStart, iLimitSwitchActive :=, iLimitSoftActive :=, iRunningTimeout := t#40s, iHomingTimeout := t#10s, iAutoPosition := "ServoV90_A4".Auto.Pos["ServoV90_A4".Auto.Index].Pos, iAutoVelocity := "ServoV90_A4".Auto.Pos["ServoV90_A4".Auto.Index].Vel, iManListPosition := "ServoV90_A4".Manual.Pos["ServoV90_A4".Manual.Index].Pos, iManListVelocity := "ServoV90_A4".Manual.Pos["ServoV90_A4".Manual.Index].Vel, iManPosition := "ServoV90_A4".In.iManPosition, iManVelocity := "ServoV90_A4".In.iManVelocity, iMode := 2, iAListNumber := "ServoV90_A4".Auto.Index, iMListNumber := "ServoV90_A4".Manual.Index, iHWIDSTW := "OP10_383A1~驱动_1~西门子报文_111__PZD-12_12", iHWIDZSW := "OP10_383A1~驱动_1~西门子报文_111__PZD-12_12", iHardwareId := "OP10_383A1~驱动_1~西门子报文_111__PZD-12_12", iSpecJog :=, iHomeSwitch :=, iIndexTableON := FALSE, Position_sensor_1 :=, Position_sensor_2 :=, Position_sensor_3 :=, Position_sensor_4 :=, "Type" :=, ioManEnale := "ServoV90_A4".IO.ioManEnale, ioAutoEnale := "ServoV90_A4".IO.ioAutoEnale, ioHome :=, ioHomeWrite :=, ioBusy :=, ioDone :=, oReady => "ServoV90_A4".Out.oReady, oWarning => "ServoV90_A4".Out.oWarning, oError => "ServoV90_A4".Out.oError, oInterlock => "ServoV90_A4".Out.oInterlock, oServoEnable => "ServoV90_A4".Out.oServoEnable, oRunning => "ServoV90_A4".Out.oRunning, oHoming => "ServoV90_A4".Out.oHoming, oHomeRef => "ServoV90_A4".Out.oHomeRef, oServoPosOK => "ServoV90_A4".Out.oServoPosOK, oErrorCode => "ServoV90_A4".Out.oErrorCode, oStatus => "ServoV90_A4".Out.oStatus, oActPosition => "ServoV90_A4".Out.oActPosition, oTargetPos =>, oPosOK => "ServoV90_A4".PositionOk, oDisable =>, oSensorInPos =>)
   END_RUNG
   // the same network as SCL:
   #Servo_383A1(iSysRun := "Station_Sys".Status.Run,   // "fbV90Ctrl"
                iReset := "Station_Sys".Cmd.Reset,
                iEstop := "Station_Sys".Status.EStopOK,
                iAuto := "Station_Sys".Auto.Mode,
                iManual := "Station_Sys".Manual.Mode,
                iConnect := true,
                iInterlock := "ServoV90_A4".In.iInterlock,
                "iManJog+" := "ServoV90_A4".In."iManJog+",
                "iManJog-" := "ServoV90_A4".In."iManJog-",
                iManStart := "ServoV90_A4".In.iManStart,
                iManListStart := "ServoV90_A4".In.iManListStart,
                iAutoStart := "ServoV90_A4".In.iAutoStart,
                iRunningTimeout := t#40s,
                iHomingTimeout := t#10s,
                iAutoPosition := "ServoV90_A4".Auto.Pos["ServoV90_A4".Auto.Index].Pos,
                iAutoVelocity := "ServoV90_A4".Auto.Pos["ServoV90_A4".Auto.Index].Vel,
                iManListPosition := "ServoV90_A4".Manual.Pos["ServoV90_A4".Manual.Index].Pos,
                iManListVelocity := "ServoV90_A4".Manual.Pos["ServoV90_A4".Manual.Index].Vel,
                iManPosition := "ServoV90_A4".In.iManPosition,
                iManVelocity := "ServoV90_A4".In.iManVelocity,
                iMode := 2,
                iAListNumber := "ServoV90_A4".Auto.Index,
                iMListNumber := "ServoV90_A4".Manual.Index,
                iHWIDSTW := "OP10_383A1~驱动_1~西门子报文_111__PZD-12_12",
                iHWIDZSW := "OP10_383A1~驱动_1~西门子报文_111__PZD-12_12",
                iHardwareId := "OP10_383A1~驱动_1~西门子报文_111__PZD-12_12",
                iIndexTableON := FALSE,
                ioManEnale := "ServoV90_A4".IO.ioManEnale,
                ioAutoEnale := "ServoV90_A4".IO.ioAutoEnale,
                oReady => "ServoV90_A4".Out.oReady,
                oWarning => "ServoV90_A4".Out.oWarning,
                oError => "ServoV90_A4".Out.oError,
                oInterlock => "ServoV90_A4".Out.oInterlock,
                oServoEnable => "ServoV90_A4".Out.oServoEnable,
                oRunning => "ServoV90_A4".Out.oRunning,
                oHoming => "ServoV90_A4".Out.oHoming,
                oHomeRef => "ServoV90_A4".Out.oHomeRef,
                oServoPosOK => "ServoV90_A4".Out.oServoPosOK,
                oErrorCode => "ServoV90_A4".Out.oErrorCode,
                oStatus => "ServoV90_A4".Out.oStatus,
                oActPosition => "ServoV90_A4".Out.oActPosition,
                oPosOK => "ServoV90_A4".PositionOk);
END_REGION

REGION Network 33 (SCL): 故障显示 / Fault indication
   //"ST70_DeviceError".Servo2.ServoDriverError := "ServoV90_A4".Out.oError;
END_REGION

REGION Network 34: *********************************伺服位置判断**********************************************
END_REGION

REGION Network 35 (SCL): 伺服位置判断 / Servo position judgment
   FOR "ServoV90_DeviceCtl".V90Servo[1].i := 1 TO 12 BY 1 DO
       "ServoV90_DeviceCtl".V90Servo[1].Pos.List["ServoV90_DeviceCtl".V90Servo[1].i].Pos := "ServoV90_A1".Auto.Pos["ServoV90_DeviceCtl".V90Servo[1].i].Pos;
       "ServoV90_DeviceCtl".V90Servo[1].Pos.List["ServoV90_DeviceCtl".V90Servo[1].i].Vel := "ServoV90_A1".Auto.Pos["ServoV90_DeviceCtl".V90Servo[1].i].Vel;

       "ServoV90_DeviceCtl".V90Servo[2].Pos.List["ServoV90_DeviceCtl".V90Servo[1].i].Pos := "ServoV90_A2".Auto.Pos["ServoV90_DeviceCtl".V90Servo[1].i].Pos;
       "ServoV90_DeviceCtl".V90Servo[2].Pos.List["ServoV90_DeviceCtl".V90Servo[1].i].Vel := "ServoV90_A2".Auto.Pos["ServoV90_DeviceCtl".V90Servo[1].i].Vel;

       "ServoV90_DeviceCtl".V90Servo[3].Pos.List["ServoV90_DeviceCtl".V90Servo[1].i].Pos := "ServoV90_A3".Auto.Pos["ServoV90_DeviceCtl".V90Servo[1].i].Pos;
       "ServoV90_DeviceCtl".V90Servo[3].Pos.List["ServoV90_DeviceCtl".V90Servo[1].i].Vel := "ServoV90_A3".Auto.Pos["ServoV90_DeviceCtl".V90Servo[1].i].Vel;

       "ServoV90_DeviceCtl".V90Servo[4].Pos.List["ServoV90_DeviceCtl".V90Servo[1].i].Pos := "ServoV90_A4".Auto.Pos["ServoV90_DeviceCtl".V90Servo[1].i].Pos;
       "ServoV90_DeviceCtl".V90Servo[4].Pos.List["ServoV90_DeviceCtl".V90Servo[1].i].Vel := "ServoV90_A4".Auto.Pos["ServoV90_DeviceCtl".V90Servo[1].i].Vel;

   END_FOR;

   (******************************************************* SV1 ********************************************************************)   
   //伺服位置判断
   #"Servo1"(iRef_Homed :=   "ServoV90_A1".Out.oHomeRef,
                             iStandstill := FALSE,
                             iReset := "Station_Sys".Cmd.Reset,
                             interlcok:="ServoV90_A1".In.iInterlock,
                             "iActual Posi" :="ServoV90_A1".Out.oActPosition,
                             "iTol+" := 50,
                             "iTol-" := 50,
                             iStartTon := T#100mS,
                             ioPoint:="ServoV90_DeviceCtl".V90Servo[1].Point,
                             oStartPos => #Sevro1StartList,
                             ioList := "ServoV90_DeviceCtl".V90Servo[1].Pos,
                             ioPosNumberSelect := "ServoV90_DeviceCtl".V90Servo[1].nPositionListNo);

   IF "ServoV90_DeviceCtl".V90Servo[1].nPositionListNo = 0 THEN
      "ServoV90_DeviceCtl".V90Servo[1].nPositionListNo:= 1 ;
   END_IF;

    //伺服位置号给定
                   // IF NOT "D-2 ModuleD-2 横向抓取移栽/拍照/旋转_IDB".伺服到下料位.X THEN
                   //     "ServoV90_A1".Auto.Index := "ServoV90_DeviceCtl".V90Servo[1].nPositionListNo;
                   // END_IF;

                  "ServoV90_A1".Auto.Index := "ServoV90_DeviceCtl".V90Servo[1].nPositionListNo;

   //伺服启动
                   "ServoV90_A1".In.iAutoStart := #Sevro1StartList;


   (******************************************************* SV2 ********************************************************************)                
   //伺服位置判断
   #"Servo2"(iRef_Homed := "ServoV90_A2".Out.oHomeRef,
             iStandstill := FALSE,
             iReset := "Station_Sys".Cmd.Reset,
             interlcok := "ServoV90_A2".In.iInterlock,
             "iActual Posi" := "ServoV90_A2".Out.oActPosition,
             "iTol+" := 50,
             "iTol-" := 50,
             iStartTon := T#100mS,
             ioPoint := "ServoV90_DeviceCtl".V90Servo[2].Point,
             oStartPos => #Sevro2StartList,
             ioList := "ServoV90_DeviceCtl".V90Servo[2].Pos,
             ioPosNumberSelect := "ServoV90_DeviceCtl".V90Servo[2].nPositionListNo);

   IF "ServoV90_DeviceCtl".V90Servo[2].nPositionListNo = 0 THEN
       "ServoV90_DeviceCtl".V90Servo[2].nPositionListNo := 1;
   END_IF;

   //伺服位置号给定
   // IF NOT "D-3 ModuleD-3从转台下料到托盘移栽机构_IDB".移栽伺服到取料位1.X THEN
   //     "ServoV90_A2".Auto.Index := "ServoV90_DeviceCtl".CMMTServo[2].nPositionListNo;
   // END_IF;

   "ServoV90_A2".Auto.Index := "ServoV90_DeviceCtl".V90Servo[2].nPositionListNo;

   //伺服启动
   "ServoV90_A2".In.iAutoStart := #Sevro2StartList;


   (******************************************************* SV3 ********************************************************************)
   //伺服位置判断
   #"Servo3"(iRef_Homed := "ServoV90_A3".Out.oHomeRef,
             iStandstill := FALSE,
             iReset := "Station_Sys".Cmd.Reset,
             interlcok := "ServoV90_A3".In.iInterlock,
             "iActual Posi" := "ServoV90_A3".Out.oActPosition,
             "iTol+" := 50,
             "iTol-" := 50,
             iStartTon := T#100mS,
             ioPoint := "ServoV90_DeviceCtl".V90Servo[3].Point,
             oStartPos => #Sevro3StartList,
             ioList := "ServoV90_DeviceCtl".V90Servo[3].Pos,
             ioPosNumberSelect := "ServoV90_DeviceCtl".V90Servo[3].nPositionListNo);

   IF "ServoV90_DeviceCtl".V90Servo[3].nPositionListNo = 0 THEN
       "ServoV90_DeviceCtl".V90Servo[3].nPositionListNo := 1;
   END_IF;
   //伺服位置号给定
   // IF NOT "D-3 ModuleD-3从转台下料到托盘移栽机构_IDB".移栽伺服到取料位1.X THEN
   //     "ServoV90_A2".Auto.Index := "ServoV90_DeviceCtl".V90Servo[2].nPositionListNo;
   // END_IF;

   "ServoV90_A3".Auto.Index := "ServoV90_DeviceCtl".V90Servo[3].nPositionListNo;

   //伺服启动
   "ServoV90_A3".In.iAutoStart := #Sevro3StartList;


   (******************************************************* SV4 ********************************************************************)
   //伺服位置判断
   #"Servo4"(iRef_Homed := "ServoV90_A4".Out.oHomeRef,
             iStandstill := FALSE,
             iReset := "Station_Sys".Cmd.Reset,
             interlcok := "ServoV90_A4".In.iInterlock,
             "iActual Posi" := "ServoV90_A4".Out.oActPosition,
             "iTol+" := 50,
             "iTol-" := 50,
             iStartTon := T#100mS,
             ioPoint := "ServoV90_DeviceCtl".V90Servo[4].Point,
             oStartPos => #Sevro4StartList,
             ioList := "ServoV90_DeviceCtl".V90Servo[4].Pos,
             ioPosNumberSelect := "ServoV90_DeviceCtl".V90Servo[4].nPositionListNo);

   IF "ServoV90_DeviceCtl".V90Servo[4].nPositionListNo = 0 THEN
       "ServoV90_DeviceCtl".V90Servo[4].nPositionListNo := 1;
   END_IF;

   //伺服位置号给定
   // IF NOT "D-3 ModuleD-3从转台下料到托盘移栽机构_IDB".移栽伺服到取料位1.X THEN
   //     "ServoV90_A2".Auto.Index := "ServoV90_DeviceCtl".V90Servo[2].nPositionListNo;
   // END_IF;

   "ServoV90_A4".Auto.Index := "ServoV90_DeviceCtl".V90Servo[4].nPositionListNo;

   //伺服启动
   "ServoV90_A4".In.iAutoStart := #Sevro4StartList;
END_REGION

REGION Network 36 (SCL): 初始化脉冲 置位手动使能 / The initial pulse set function was manually enabled
   IF "FirstScan" THEN
       "ServoV90_A1".IO.ioManEnale := TRUE;
       "ServoV90_A2".IO.ioManEnale := TRUE;
       "ServoV90_A3".IO.ioManEnale := TRUE;
       "ServoV90_A4".IO.ioManEnale := TRUE;
   END_IF;
END_REGION
END_FUNCTION_BLOCK

FUNCTION_BLOCK "fbV90Ctrl"   // FB1820, LAD
{ S7_Optimized_Access := 'FALSE' }
// stored: AutoNumber false, SetENOAutomatically false
   VAR_INPUT
      iSysRun : Bool := false;   // PowerOn
      iReset : Bool := false;   // reset action
      iEstop : Bool := false;
      iAuto : Bool := false;   // auto mode
      iManual : Bool := false;   // manual mode
      iConnect : Bool := false;   // Bus status
      iStep : Bool := false;   // step mode
      iInterlock : Bool := false;   // interlock
      "iManJog+" : Bool := false;   // positive motion/action/...manually
      "iManJog-" : Bool := false;   // negtive motion/action/...manually
      iManStart : Bool := false;   // positive motion/action/...automaticly
      iManListStart : Bool := false;
      iAutoStart : Bool := false;   // negtive motion/action/...automaticly
      iLimitSwitchActive : Bool := true;   // hardware limit switch active
      iLimitSoftActive : Bool := true;   // Soft limit active
      iRunningTimeout : Time := T#0ms;
      iHomingTimeout : Time := T#0ms;
      iAutoPosition : DInt := 0;
      iAutoVelocity : Int := 0;
      iManListPosition : DInt := 0;
      iManListVelocity : Int := 0;
      iManPosition : DInt := 0;
      iManVelocity : Int := 0;
      iMode : Int := 0;   // 1-相对;2-绝对
      iAListNumber : Int := 0;   // 当前列表程序号
      iMListNumber : Int := 0;   // 当前列表程序号
      iHWIDSTW : HW_IO := 0;   // CMMT 设备视图111报文硬件标识符 Send
      iHWIDZSW : HW_IO := 0;   // CMMT 设备视图111报文硬件标识符 Recive
      iHardwareId : HW_IO := 0;
      iSpecJog : Bool := false;   // 自动下jog
      iHomeSwitch : Bool := false;   // 原点开关
      iIndexTableON : Bool := false;   // 转台激活
      Position_sensor_1 : Bool := false;
      Position_sensor_2 : Bool := false;
      Position_sensor_3 : Bool := false;
      Position_sensor_4 : Bool := false;
      "Type" : Bool;   // =0:窄产品，=1:宽产品
   END_VAR
   VAR_OUTPUT
      oReady : Bool;
      oWarning : Bool;   // warning
      oError : Bool;   // error
      oInterlock : Bool;
      oServoEnable : Bool;
      oRunning : Bool;
      oHoming : Bool;
      oHomeRef : Bool;
      oServoPosOK : Bool;
      oErrorCode : Int;
      oStatus : Int;
      oActPosition : DInt;
      oTargetPos : DInt;
      oPosOK : Array[1..20] of Bool;
      oDisable : Bool;
      oSensorInPos : Bool;   // 传感器检测在位置上
   END_VAR
   VAR_IN_OUT
      ioManEnale : Bool;
      ioAutoEnale : Bool;
      ioHome : Bool;
      ioHomeWrite : Bool;
      ioBusy : Bool;
      ioDone : Bool;
   END_VAR
   VAR
      sStep : Array[1..4] of Int;
      sPls : Array[1..16] of Bool;
      sErrorCode : Int;
      sPosOK : Bool;
      sRunning : Bool;
      sHoming : Bool;
      sCancel : Bool;
      "sMan/List" : Bool;   // 0-manual input;1-manual listmode
      sCMMT { S7_SetPoint := 'True'} : "SINA_POS";
      sPara { S7_SetPoint := 'True'} : "SINA_PARA_S";
      sRunningTimeout { S7_SetPoint := 'True'} : TON_TIME;
      sHomingTimeout { S7_SetPoint := 'True'} : TON_TIME;
      sEnableDelay { S7_SetPoint := 'True'} : TON_TIME;
      sManDirHis : DInt;
      sManListHis : Int;
      sAutoListHis : Int;
      Position_PV : Int;   // 实际位置
      Conv_Pos_PV : Int;   // 转换后位置
      Delay : TON_TIME;
      Delay_1 : TON_TIME;
      Delay_2 { S7_SetPoint := 'True'} : TON_TIME;
      Delay_3 { S7_SetPoint := 'True'} : TON_TIME;
   END_VAR
   VAR_TEMP
      tNormalON : Bool;
      tHome : Bool;   // Homing
      tCancelTask : Bool;   // Cancel task
      tPauseTask : Bool;   // Pause task
      tRetVal : Int;
      "tPosConfig+" : DInt;
      "tPosConfig-" : DInt;
   END_VAR
   VAR CONSTANT
      cOffset : DInt := 20;
   END_VAR
   VAR_TEMP   // added for the SCL form of the ladder/FBD networks
      _w1 : Bool;
      _w2 : Bool;
      _w3 : Bool;
      _w4 : Bool;
      _w5 : Bool;
      _w6 : Bool;
      _w7 : Bool;
      _w8 : Bool;
      _w9 : Bool;
      _w10 : Bool;
      _w11 : Bool;
      _w12 : Bool;
      _w13 : Bool;
   END_VAR
BEGIN

REGION Network 1
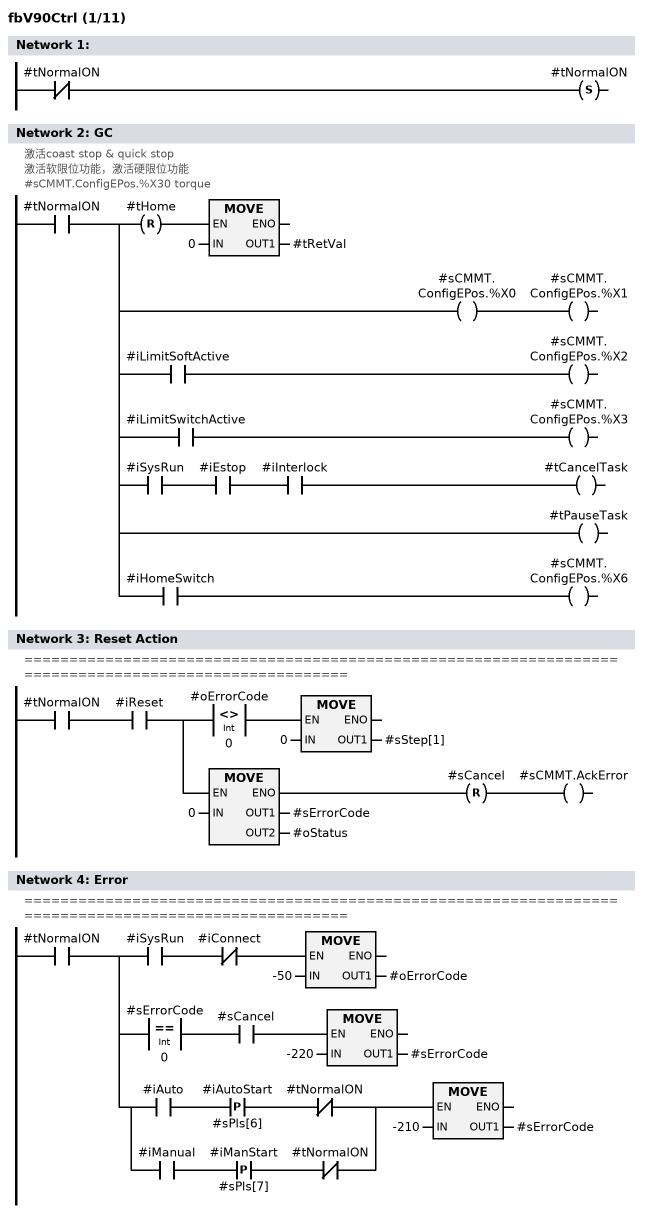
   RUNG wire#powerrail
      I_Contact( #tNormalON )
      S_Coil( #tNormalON )
   END_RUNG
   // the same network as SCL:
   IF NOT #tNormalON THEN #tNormalON := TRUE; END_IF;
END_REGION

REGION Network 2: GC
   // 激活coast stop & quick stop 
   // 激活软限位功能，激活硬限位功能
   // #sCMMT.ConfigEPos.%X30 torque
   RUNG wire#powerrail
      Contact( #tNormalON )
      wire#w1
      R_Coil( #tHome )
      Move(in := 0, out1 => #tRetVal)
   END_RUNG
   RUNG wire#w1
      Coil( #sCMMT.ConfigEPos.%X0 )
      Coil( #sCMMT.ConfigEPos.%X1 )
   END_RUNG
   RUNG wire#w1
      Contact( #iLimitSoftActive )
      Coil( #sCMMT.ConfigEPos.%X2 )
   END_RUNG
   RUNG wire#w1
      Contact( #iLimitSwitchActive )
      Coil( #sCMMT.ConfigEPos.%X3 )
   END_RUNG
   RUNG wire#w1
      Contact( #iSysRun )
      Contact( #iEstop )
      Contact( #iInterlock )
      Coil( #tCancelTask )
   END_RUNG
   RUNG wire#w1
      Coil( #tPauseTask )
   END_RUNG
   RUNG wire#w1
      Contact( #iHomeSwitch )
      Coil( #sCMMT.ConfigEPos.%X6 )
   END_RUNG
   // the same network as SCL:
   IF #tNormalON THEN
       #tHome := FALSE;
       #tRetVal := 0;
   END_IF;
   #sCMMT.ConfigEPos.%X0 := #tNormalON;
   #sCMMT.ConfigEPos.%X1 := #tNormalON;
   #sCMMT.ConfigEPos.%X2 := #tNormalON AND #iLimitSoftActive;
   #sCMMT.ConfigEPos.%X3 := #tNormalON AND #iLimitSwitchActive;
   #tCancelTask := #tNormalON AND #iSysRun AND #iEstop AND #iInterlock;
   #tPauseTask := #tNormalON;
   #sCMMT.ConfigEPos.%X6 := #tNormalON AND #iHomeSwitch;
END_REGION

REGION Network 3: Reset Action
   // ======================================================================================================
   RUNG wire#powerrail
      Contact( #tNormalON )
      Contact( #iReset )
      wire#w1
      { S7_Templates := "SrcType := Int" } NE_Contact(in1 := #oErrorCode, in2 := 0)
      Move(in := 0, out1 => #sStep[1])
   END_RUNG
   RUNG wire#w1
      Move(in := 0, out1 => #sErrorCode, out2 => #oStatus)
      R_Coil( #sCancel )
      Coil( #sCMMT.AckError )
   END_RUNG
   // the same network as SCL:
   #_w1 := #tNormalON AND #iReset;
   IF #_w1 AND (#oErrorCode <> 0) THEN #sStep[1] := 0; END_IF;
   IF #_w1 THEN
       #sErrorCode := 0;
       #oStatus := 0;
       #sCancel := FALSE;
   END_IF;
   #sCMMT.AckError := #_w1;
END_REGION

REGION Network 4: Error
   // ======================================================================================================
   RUNG wire#powerrail
      Contact( #tNormalON )
      wire#w1
      Contact( #iSysRun )
      I_Contact( #iConnect )
      Move(in := -50, out1 => #oErrorCode)
   END_RUNG
   RUNG wire#w1
      { S7_Templates := "SrcType := Int" } EQ_Contact(in1 := #sErrorCode, in2 := 0)
      Contact( #sCancel )
      Move(in := -220, out1 => #sErrorCode)
   END_RUNG
   RUNG wire#w1
      Contact( #iAuto )
      P_Contact(operand := #iAutoStart, bit := #sPls[6])
      I_Contact( #tNormalON )
      wire#w2
      Move(in := -210, out1 => #sErrorCode)
   END_RUNG
   RUNG wire#w1
      Contact( #iManual )
      P_Contact(operand := #iManStart, bit := #sPls[7])
      I_Contact( #tNormalON )
   END_RUNG wire#w2
   // the same network as SCL:
   IF #tNormalON AND #iSysRun AND NOT #iConnect THEN #oErrorCode := -50; END_IF;
   IF #tNormalON AND (#sErrorCode = 0) AND #sCancel THEN #sErrorCode := -220; END_IF;
   #_w1 := #tNormalON AND #iAuto AND #iAutoStart AND NOT #sPls[6];   // rising edge of #iAutoStart
   #sPls[6] := #iAutoStart;
   #_w2 := #tNormalON AND #iManual AND #iManStart AND NOT #sPls[7];   // rising edge of #iManStart
   #sPls[7] := #iManStart;
   IF (#_w1 AND NOT #tNormalON) OR (#_w2 AND NOT #tNormalON) THEN #sErrorCode := -210; END_IF;
END_REGION

REGION Network 5: preCondition
   // #sCMMT.EnableAxis  使能驱动器
   // 设备打到自动模式下就将手动使能复位
   // ================================
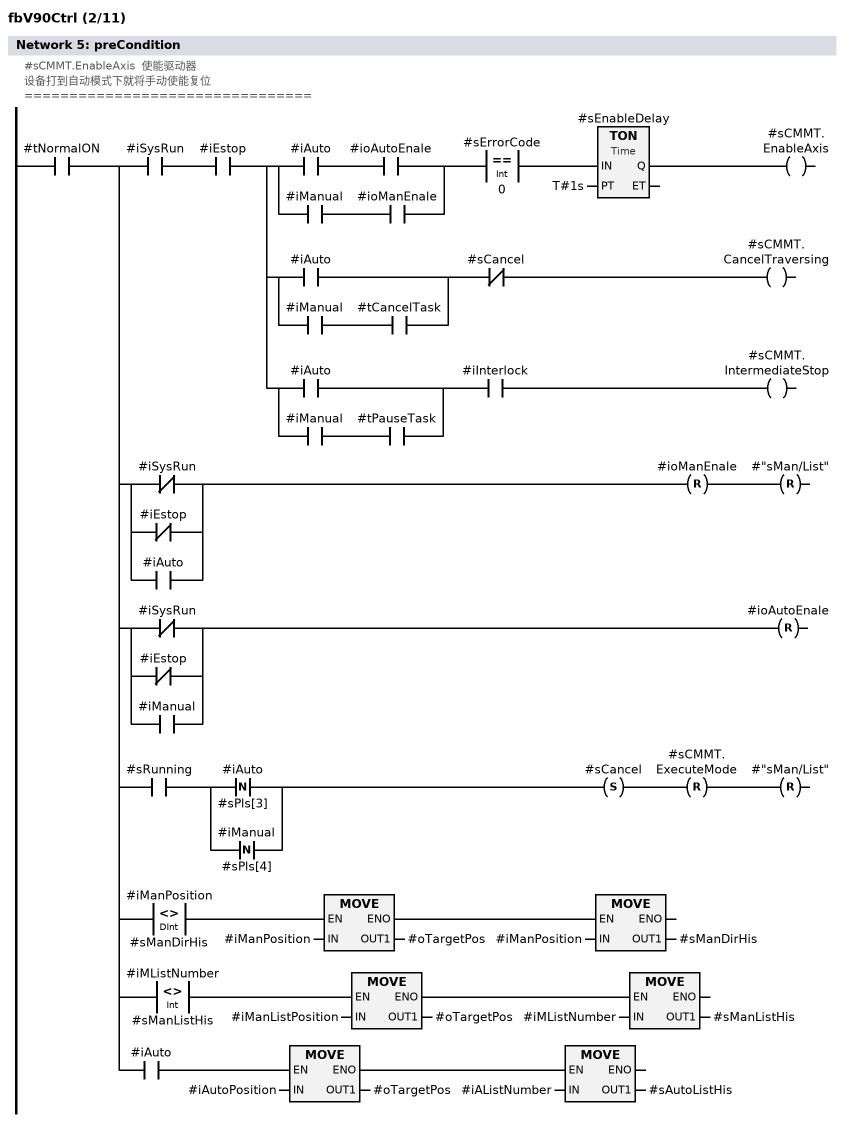
   RUNG wire#powerrail
      Contact( #tNormalON )
      wire#w1
      Contact( #iSysRun )
      Contact( #iEstop )
      wire#w2
      Contact( #iAuto )
      Contact( #ioAutoEnale )
      wire#w3
      { S7_Templates := "SrcType := Int" } EQ_Contact(in1 := #sErrorCode, in2 := 0)
      { S7_Templates := "time_type := Time" } #sEnableDelay.TON(pt := T#1s, et =>)
      Coil( #sCMMT.EnableAxis )
   END_RUNG
   RUNG wire#w2
      Contact( #iManual )
      Contact( #ioManEnale )
   END_RUNG wire#w3
   RUNG wire#w2
      Contact( #iAuto )
      wire#w4
      I_Contact( #sCancel )
      Coil( #sCMMT.CancelTraversing )
   END_RUNG
   RUNG wire#w2
      Contact( #iManual )
      Contact( #tCancelTask )
   END_RUNG wire#w4
   RUNG wire#w2
      Contact( #iAuto )
      wire#w5
      Contact( #iInterlock )
      Coil( #sCMMT.IntermediateStop )
   END_RUNG
   RUNG wire#w2
      Contact( #iManual )
      Contact( #tPauseTask )
   END_RUNG wire#w5
   RUNG wire#w1
      I_Contact( #iSysRun )
      wire#w6
      R_Coil( #ioManEnale )
      R_Coil( #"sMan/List" )
   END_RUNG
   RUNG wire#w1
      I_Contact( #iEstop )
   END_RUNG wire#w6
   RUNG wire#w1
      Contact( #iAuto )
   END_RUNG wire#w6
   RUNG wire#w1
      I_Contact( #iSysRun )
      wire#w7
      R_Coil( #ioAutoEnale )
   END_RUNG
   RUNG wire#w1
      I_Contact( #iEstop )
   END_RUNG wire#w7
   RUNG wire#w1
      Contact( #iManual )
   END_RUNG wire#w7
   RUNG wire#w1
      Contact( #sRunning )
      wire#w8
      N_Contact(operand := #iAuto, bit := #sPls[3])
      wire#w9
      S_Coil( #sCancel )
      R_Coil( #sCMMT.ExecuteMode )
      R_Coil( #"sMan/List" )
   END_RUNG
   RUNG wire#w8
      N_Contact(operand := #iManual, bit := #sPls[4])
   END_RUNG wire#w9
   RUNG wire#w1
      { S7_Templates := "SrcType := DInt" } NE_Contact(in1 := #iManPosition, in2 := #sManDirHis)
      Move(in := #iManPosition, out1 => #oTargetPos)
      Move(in := #iManPosition, out1 => #sManDirHis)
   END_RUNG
   RUNG wire#w1
      { S7_Templates := "SrcType := Int" } NE_Contact(in1 := #iMListNumber, in2 := #sManListHis)
      Move(in := #iManListPosition, out1 => #oTargetPos)
      Move(in := #iMListNumber, out1 => #sManListHis)
   END_RUNG
   RUNG wire#w1
      Contact( #iAuto )
      Move(in := #iAutoPosition, out1 => #oTargetPos)
      Move(in := #iAListNumber, out1 => #sAutoListHis)
   END_RUNG
   // the same network as SCL:
   #_w1 := #tNormalON AND #iSysRun AND #iEstop;
   #sEnableDelay(IN := #_w1 AND ((#iAuto AND #ioAutoEnale) OR (#iManual AND #ioManEnale)) AND (#sErrorCode = 0),   // TON
                 PT := T#1s);
   #sCMMT.EnableAxis := #sEnableDelay.Q;
   #sCMMT.CancelTraversing := #_w1 AND (#iAuto OR (#iManual AND #tCancelTask)) AND NOT #sCancel;
   #sCMMT.IntermediateStop := #_w1 AND (#iAuto OR (#iManual AND #tPauseTask)) AND #iInterlock;
   IF #tNormalON AND (NOT #iSysRun OR NOT #iEstop OR #iAuto) THEN
       #ioManEnale := FALSE;
       #"sMan/List" := FALSE;
   END_IF;
   IF #tNormalON AND (NOT #iSysRun OR NOT #iEstop OR #iManual) THEN #ioAutoEnale := FALSE; END_IF;
   #_w2 := #tNormalON AND #sRunning AND NOT #iAuto AND #sPls[3];   // falling edge of #iAuto
   #sPls[3] := #iAuto;
   #_w3 := #tNormalON AND #sRunning AND NOT #iManual AND #sPls[4];   // falling edge of #iManual
   #sPls[4] := #iManual;
   IF #_w2 OR #_w3 THEN
       #sCancel := TRUE;
       #sCMMT.ExecuteMode := FALSE;
       #"sMan/List" := FALSE;
   END_IF;
   IF #tNormalON AND (#iManPosition <> #sManDirHis) THEN
       #oTargetPos := #iManPosition;
       #sManDirHis := #iManPosition;
   END_IF;
   IF #tNormalON AND (#iMListNumber <> #sManListHis) THEN
       #oTargetPos := #iManListPosition;
       #sManListHis := #iMListNumber;
   END_IF;
   IF #tNormalON AND #iAuto THEN
       #oTargetPos := #iAutoPosition;
       #sAutoListHis := #iAListNumber;
   END_IF;
END_REGION

REGION Network 6: JOG+&JOG-
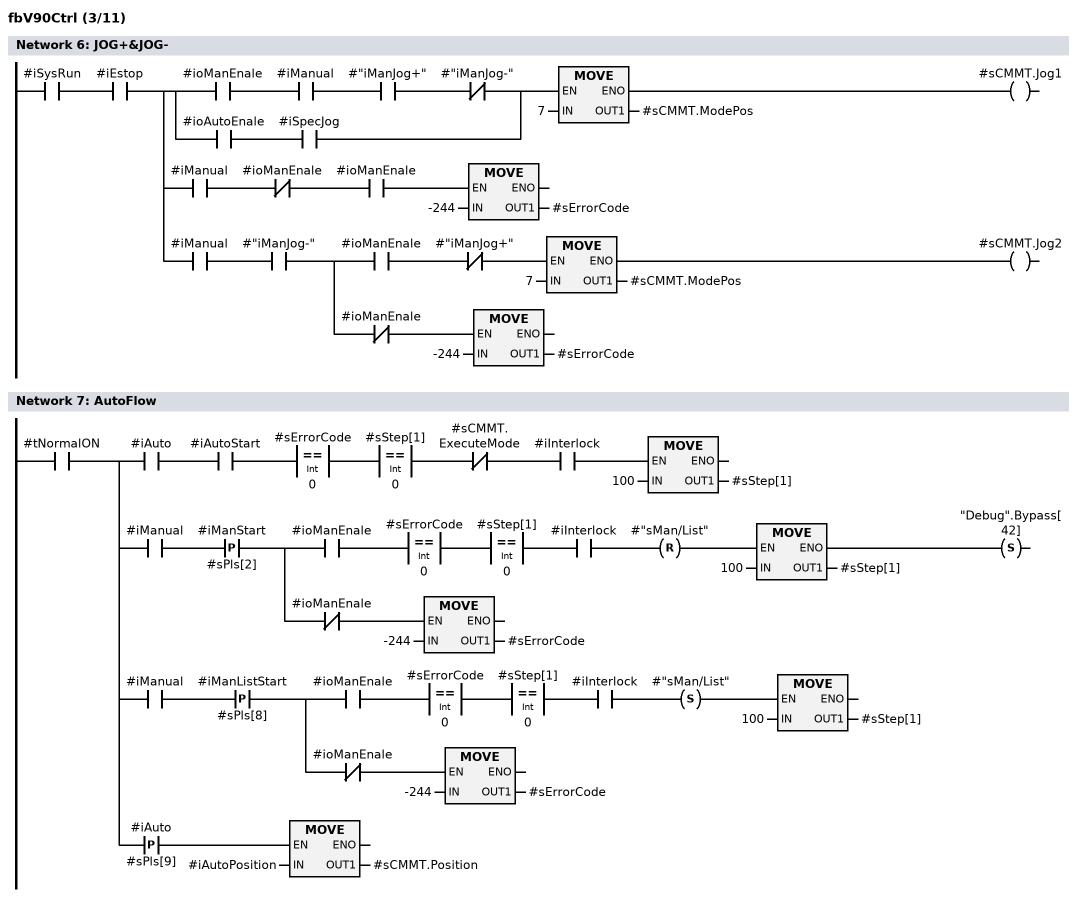
   RUNG wire#powerrail
      Contact( #iSysRun )
      Contact( #iEstop )
      wire#w1
      Contact( #ioManEnale )
      Contact( #iManual )
      Contact( #"iManJog+" )
      I_Contact( #"iManJog-" )
      wire#w2
      Move(in := 7, out1 => #sCMMT.ModePos)
      Coil( #sCMMT.Jog1 )
   END_RUNG
   RUNG wire#w1
      Contact( #ioAutoEnale )
      Contact( #iSpecJog )
   END_RUNG wire#w2
   RUNG wire#w1
      Contact( #iManual )
      I_Contact( #ioManEnale )
      Contact( #ioManEnale )
      Move(in := -244, out1 => #sErrorCode)
   END_RUNG
   RUNG wire#w1
      Contact( #iManual )
      Contact( #"iManJog-" )
      wire#w3
      Contact( #ioManEnale )
      I_Contact( #"iManJog+" )
      Move(in := 7, out1 => #sCMMT.ModePos)
      Coil( #sCMMT.Jog2 )
   END_RUNG
   RUNG wire#w3
      I_Contact( #ioManEnale )
      Move(in := -244, out1 => #sErrorCode)
   END_RUNG
   // the same network as SCL:
   #_w1 := #iSysRun AND #iEstop;
   #_w2 := #_w1 AND ((#ioManEnale AND #iManual AND #"iManJog+" AND NOT #"iManJog-") OR (#ioAutoEnale AND #iSpecJog));
   IF #_w2 THEN #sCMMT.ModePos := 7; END_IF;
   #sCMMT.Jog1 := #_w2;
   IF #_w1 AND #iManual AND NOT #ioManEnale AND #ioManEnale THEN #sErrorCode := -244; END_IF;
   #_w3 := #_w1 AND #iManual AND #"iManJog-";
   #_w4 := #_w3 AND #ioManEnale AND NOT #"iManJog+";
   IF #_w4 THEN #sCMMT.ModePos := 7; END_IF;
   #sCMMT.Jog2 := #_w4;
   IF #_w3 AND NOT #ioManEnale THEN #sErrorCode := -244; END_IF;
END_REGION

REGION Network 7: AutoFlow
   RUNG wire#powerrail
      Contact( #tNormalON )
      wire#w1
      Contact( #iAuto )
      Contact( #iAutoStart )
      { S7_Templates := "SrcType := Int" } EQ_Contact(in1 := #sErrorCode, in2 := 0)
      { S7_Templates := "SrcType := Int" } EQ_Contact(in1 := #sStep[1], in2 := 0)
      I_Contact( #sCMMT.ExecuteMode )
      Contact( #iInterlock )
      Move(in := 100, out1 => #sStep[1])
   END_RUNG
   RUNG wire#w1
      Contact( #iManual )
      P_Contact(operand := #iManStart, bit := #sPls[2])
      wire#w2
      Contact( #ioManEnale )
      { S7_Templates := "SrcType := Int" } EQ_Contact(in1 := #sErrorCode, in2 := 0)
      { S7_Templates := "SrcType := Int" } EQ_Contact(in1 := #sStep[1], in2 := 0)
      Contact( #iInterlock )
      R_Coil( #"sMan/List" )
      Move(in := 100, out1 => #sStep[1])
      S_Coil( "Debug".Bypass[42] )
   END_RUNG
   RUNG wire#w2
      I_Contact( #ioManEnale )
      Move(in := -244, out1 => #sErrorCode)
   END_RUNG
   RUNG wire#w1
      Contact( #iManual )
      P_Contact(operand := #iManListStart, bit := #sPls[8])
      wire#w3
      Contact( #ioManEnale )
      { S7_Templates := "SrcType := Int" } EQ_Contact(in1 := #sErrorCode, in2 := 0)
      { S7_Templates := "SrcType := Int" } EQ_Contact(in1 := #sStep[1], in2 := 0)
      Contact( #iInterlock )
      S_Coil( #"sMan/List" )
      Move(in := 100, out1 => #sStep[1])
   END_RUNG
   RUNG wire#w3
      I_Contact( #ioManEnale )
      Move(in := -244, out1 => #sErrorCode)
   END_RUNG
   RUNG wire#w1
      P_Contact(operand := #iAuto, bit := #sPls[9])
      Move(in := #iAutoPosition, out1 => #sCMMT.Position)
   END_RUNG
   // the same network as SCL:
   IF #tNormalON AND #iAuto AND #iAutoStart AND (#sErrorCode = 0) AND (#sStep[1] = 0) AND NOT #sCMMT.ExecuteMode AND #iInterlock THEN
       #sStep[1] := 100;
   END_IF;
   #_w1 := #tNormalON AND #iManual AND #iManStart AND NOT #sPls[2];   // rising edge of #iManStart
   #sPls[2] := #iManStart;
   IF #_w1 AND #ioManEnale AND (#sErrorCode = 0) AND (#sStep[1] = 0) AND #iInterlock THEN
       #"sMan/List" := FALSE;
   END_IF;
   #_w2 := #_w1 AND #ioManEnale AND (#sErrorCode = 0) AND (#sStep[1] = 0) AND #iInterlock;
   IF #_w2 THEN
       #sStep[1] := 100;
       "Debug".Bypass[42] := TRUE;
   END_IF;
   IF #_w1 AND NOT #ioManEnale THEN #sErrorCode := -244; END_IF;
   #_w3 := #tNormalON AND #iManual AND #iManListStart AND NOT #sPls[8];   // rising edge of #iManListStart
   #sPls[8] := #iManListStart;
   IF #_w3 AND #ioManEnale AND (#sErrorCode = 0) AND (#sStep[1] = 0) AND #iInterlock THEN
       #"sMan/List" := TRUE;
       #sStep[1] := 100;
   END_IF;
   IF #_w3 AND NOT #ioManEnale THEN #sErrorCode := -244; END_IF;
   #_w4 := #tNormalON AND #iAuto AND NOT #sPls[9];   // rising edge of #iAuto
   #sPls[9] := #iAuto;
   IF #_w4 THEN #sCMMT.Position := #iAutoPosition; END_IF;
END_REGION

REGION Network 8: AutoRunning
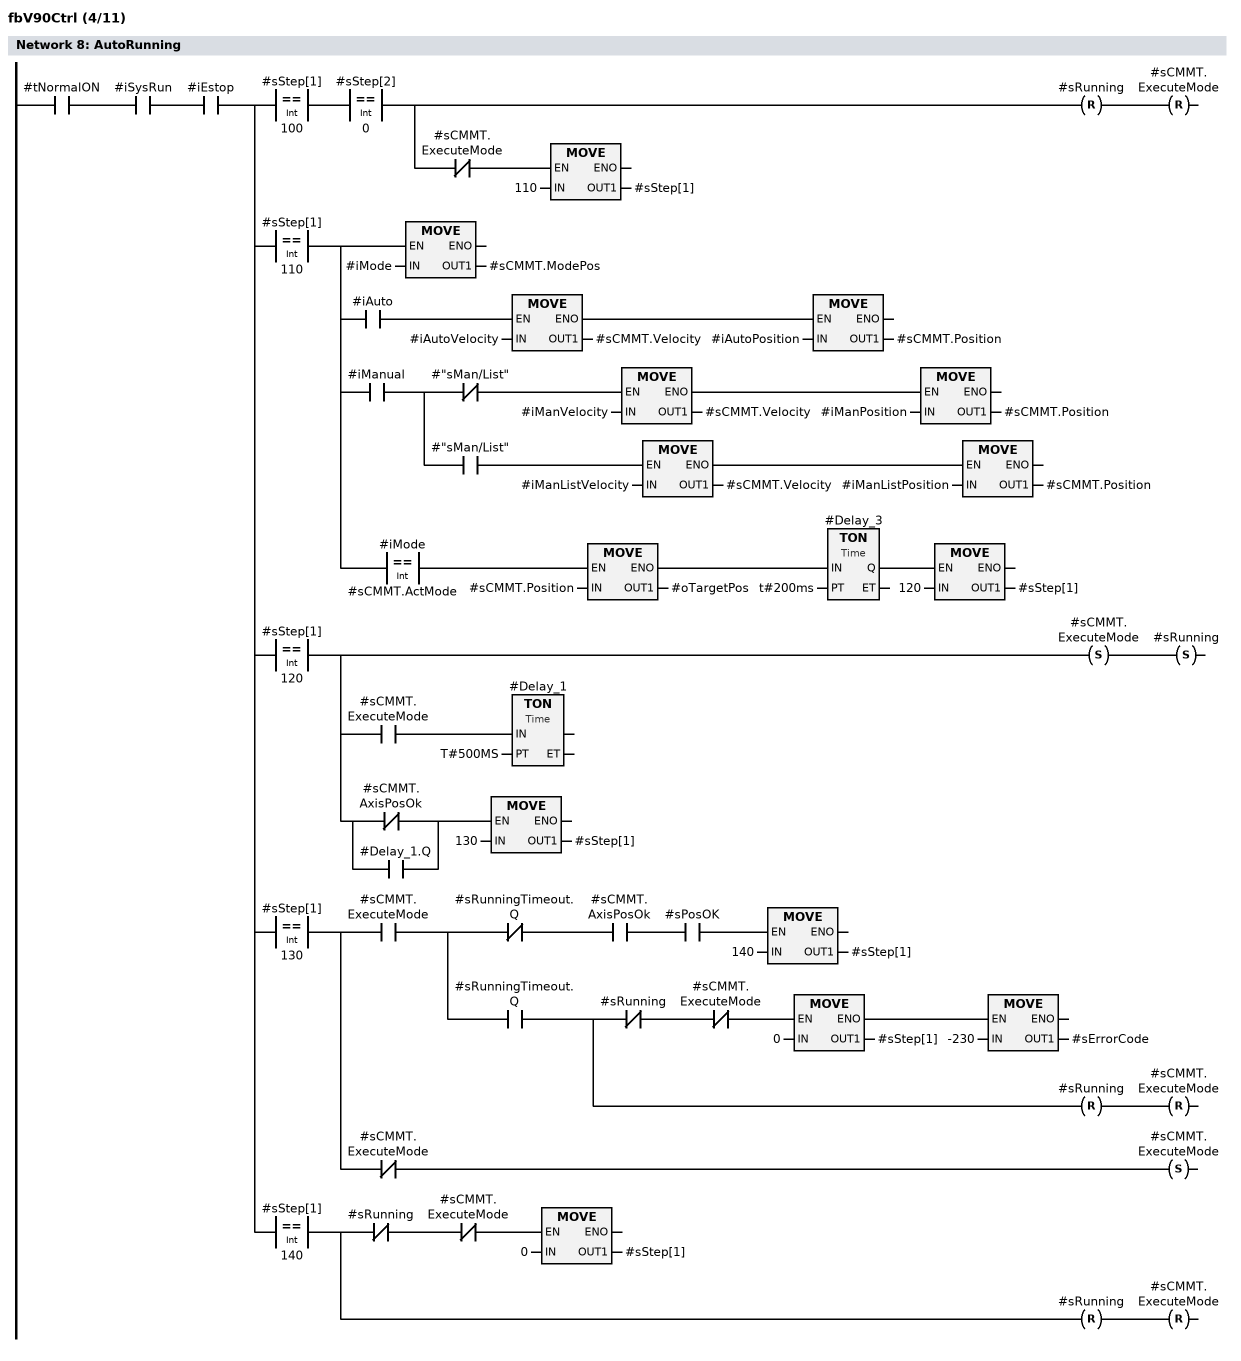
   RUNG wire#powerrail
      Contact( #tNormalON )
      Contact( #iSysRun )
      Contact( #iEstop )
      wire#w1
      { S7_Templates := "SrcType := Int" } EQ_Contact(in1 := #sStep[1], in2 := 100)
      { S7_Templates := "SrcType := Int" } EQ_Contact(in1 := #sStep[2], in2 := 0)
      wire#w2
      R_Coil( #sRunning )
      R_Coil( #sCMMT.ExecuteMode )
   END_RUNG
   RUNG wire#w2
      I_Contact( #sCMMT.ExecuteMode )
      Move(in := 110, out1 => #sStep[1])
   END_RUNG
   RUNG wire#w1
      { S7_Templates := "SrcType := Int" } EQ_Contact(in1 := #sStep[1], in2 := 110)
      wire#w3
      Move(in := #iMode, out1 => #sCMMT.ModePos)
   END_RUNG
   RUNG wire#w3
      Contact( #iAuto )
      Move(in := #iAutoVelocity, out1 => #sCMMT.Velocity)
      Move(in := #iAutoPosition, out1 => #sCMMT.Position)
   END_RUNG
   RUNG wire#w3
      Contact( #iManual )
      wire#w4
      I_Contact( #"sMan/List" )
      Move(in := #iManVelocity, out1 => #sCMMT.Velocity)
      Move(in := #iManPosition, out1 => #sCMMT.Position)
   END_RUNG
   RUNG wire#w4
      Contact( #"sMan/List" )
      Move(in := #iManListVelocity, out1 => #sCMMT.Velocity)
      Move(in := #iManListPosition, out1 => #sCMMT.Position)
   END_RUNG
   RUNG wire#w3
      { S7_Templates := "SrcType := Int" } EQ_Contact(in1 := #iMode, in2 := #sCMMT.ActMode)
      Move(in := #sCMMT.Position, out1 => #oTargetPos)
      { S7_Templates := "time_type := Time" } #Delay_3.TON(pt := t#200ms, et =>)
      Move(in := 120, out1 => #sStep[1])
   END_RUNG
   RUNG wire#w1
      { S7_Templates := "SrcType := Int" } EQ_Contact(in1 := #sStep[1], in2 := 120)
      wire#w5
      S_Coil( #sCMMT.ExecuteMode )
      S_Coil( #sRunning )
   END_RUNG
   RUNG wire#w5
      Contact( #sCMMT.ExecuteMode )
      { S7_Templates := "time_type := Time" } #Delay_1.TON(pt := T#500MS, et =>)
   END_RUNG
   RUNG wire#w5
      I_Contact( #sCMMT.AxisPosOk )
      wire#w6
      Move(in := 130, out1 => #sStep[1])
   END_RUNG
   RUNG wire#w5
      Contact( #Delay_1.Q )
   END_RUNG wire#w6
   RUNG wire#w1
      { S7_Templates := "SrcType := Int" } EQ_Contact(in1 := #sStep[1], in2 := 130)
      wire#w7
      Contact( #sCMMT.ExecuteMode )
      wire#w8
      I_Contact( #sRunningTimeout.Q )
      Contact( #sCMMT.AxisPosOk )
      Contact( #sPosOK )
      Move(in := 140, out1 => #sStep[1])
   END_RUNG
   RUNG wire#w8
      Contact( #sRunningTimeout.Q )
      wire#w9
      I_Contact( #sRunning )
      I_Contact( #sCMMT.ExecuteMode )
      Move(in := 0, out1 => #sStep[1])
      Move(in := -230, out1 => #sErrorCode)
   END_RUNG
   RUNG wire#w9
      R_Coil( #sRunning )
      R_Coil( #sCMMT.ExecuteMode )
   END_RUNG
   RUNG wire#w7
      I_Contact( #sCMMT.ExecuteMode )
      S_Coil( #sCMMT.ExecuteMode )
   END_RUNG
   RUNG wire#w1
      { S7_Templates := "SrcType := Int" } EQ_Contact(in1 := #sStep[1], in2 := 140)
      wire#w10
      I_Contact( #sRunning )
      I_Contact( #sCMMT.ExecuteMode )
      Move(in := 0, out1 => #sStep[1])
   END_RUNG
   RUNG wire#w10
      R_Coil( #sRunning )
      R_Coil( #sCMMT.ExecuteMode )
   END_RUNG
   // the same network as SCL:
   #_w1 := #tNormalON AND #iSysRun AND #iEstop;
   #_w2 := #_w1 AND (#sStep[1] = 100) AND (#sStep[2] = 0);
   IF #_w2 THEN
       #sRunning := FALSE;
       #sCMMT.ExecuteMode := FALSE;
   END_IF;
   IF #_w2 AND NOT #sCMMT.ExecuteMode THEN #sStep[1] := 110; END_IF;
   #_w3 := #_w1 AND (#sStep[1] = 110);
   IF #_w3 THEN #sCMMT.ModePos := #iMode; END_IF;
   IF #_w3 AND #iAuto THEN
       #sCMMT.Velocity := #iAutoVelocity;
       #sCMMT.Position := #iAutoPosition;
   END_IF;
   #_w4 := #_w3 AND #iManual;
   IF #_w4 AND NOT #"sMan/List" THEN
       #sCMMT.Velocity := #iManVelocity;
       #sCMMT.Position := #iManPosition;
   END_IF;
   IF #_w4 AND #"sMan/List" THEN
       #sCMMT.Velocity := #iManListVelocity;
       #sCMMT.Position := #iManListPosition;
   END_IF;
   #_w5 := #_w3 AND (#iMode = #sCMMT.ActMode);
   IF #_w5 THEN #oTargetPos := #sCMMT.Position; END_IF;
   #Delay_3(IN := #_w5, PT := t#200ms);   // TON
   IF #Delay_3.Q THEN #sStep[1] := 120; END_IF;
   #_w6 := #_w1 AND (#sStep[1] = 120);
   IF #_w6 THEN
       #sCMMT.ExecuteMode := TRUE;
       #sRunning := TRUE;
   END_IF;
   #Delay_1(IN := #_w6 AND #sCMMT.ExecuteMode, PT := T#500MS);   // TON
   IF #_w6 AND (NOT #sCMMT.AxisPosOk OR #Delay_1.Q) THEN #sStep[1] := 130; END_IF;
   #_w7 := #_w1 AND (#sStep[1] = 130);
   #_w8 := #_w7 AND #sCMMT.ExecuteMode;
   IF #_w8 AND NOT #sRunningTimeout.Q AND #sCMMT.AxisPosOk AND #sPosOK THEN #sStep[1] := 140; END_IF;
   #_w9 := #_w8 AND #sRunningTimeout.Q;
   IF #_w9 AND NOT #sRunning AND NOT #sCMMT.ExecuteMode THEN
       #sStep[1] := 0;
       #sErrorCode := -230;
   END_IF;
   IF #_w9 THEN
       #sRunning := FALSE;
       #sCMMT.ExecuteMode := FALSE;
   END_IF;
   IF #_w7 AND NOT #sCMMT.ExecuteMode THEN #sCMMT.ExecuteMode := TRUE; END_IF;
   #_w10 := #_w1 AND (#sStep[1] = 140);
   IF #_w10 AND NOT #sRunning AND NOT #sCMMT.ExecuteMode THEN #sStep[1] := 0; END_IF;
   IF #_w10 THEN
       #sRunning := FALSE;
       #sCMMT.ExecuteMode := FALSE;
   END_IF;
END_REGION

REGION Network 9: runnint timeout
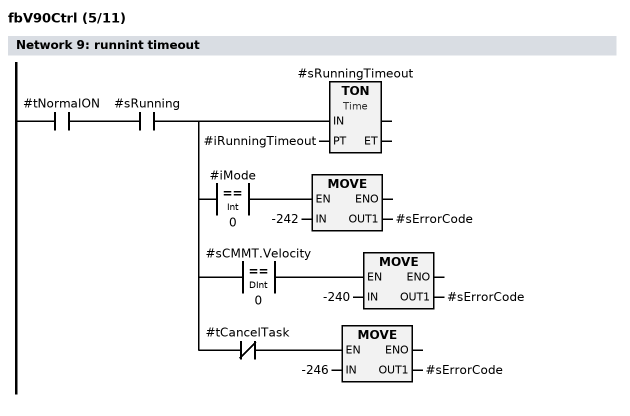
   RUNG wire#powerrail
      Contact( #tNormalON )
      Contact( #sRunning )
      wire#w1
      { S7_Templates := "time_type := Time" } #sRunningTimeout.TON(pt := #iRunningTimeout, et =>)
   END_RUNG
   RUNG wire#w1
      { S7_Templates := "SrcType := Int" } EQ_Contact(in1 := #iMode, in2 := 0)
      Move(in := -242, out1 => #sErrorCode)
   END_RUNG
   RUNG wire#w1
      { S7_Templates := "SrcType := DInt" } EQ_Contact(in1 := #sCMMT.Velocity, in2 := 0)
      Move(in := -240, out1 => #sErrorCode)
   END_RUNG
   RUNG wire#w1
      I_Contact( #tCancelTask )
      Move(in := -246, out1 => #sErrorCode)
   END_RUNG
   // the same network as SCL:
   #_w1 := #tNormalON AND #sRunning;
   #sRunningTimeout(IN := #_w1, PT := #iRunningTimeout);   // TON
   IF #_w1 AND (#iMode = 0) THEN #sErrorCode := -242; END_IF;
   IF #_w1 AND (#sCMMT.Velocity = 0) THEN #sErrorCode := -240; END_IF;
   IF #_w1 AND NOT #tCancelTask THEN #sErrorCode := -246; END_IF;
END_REGION

REGION Network 10: Homing
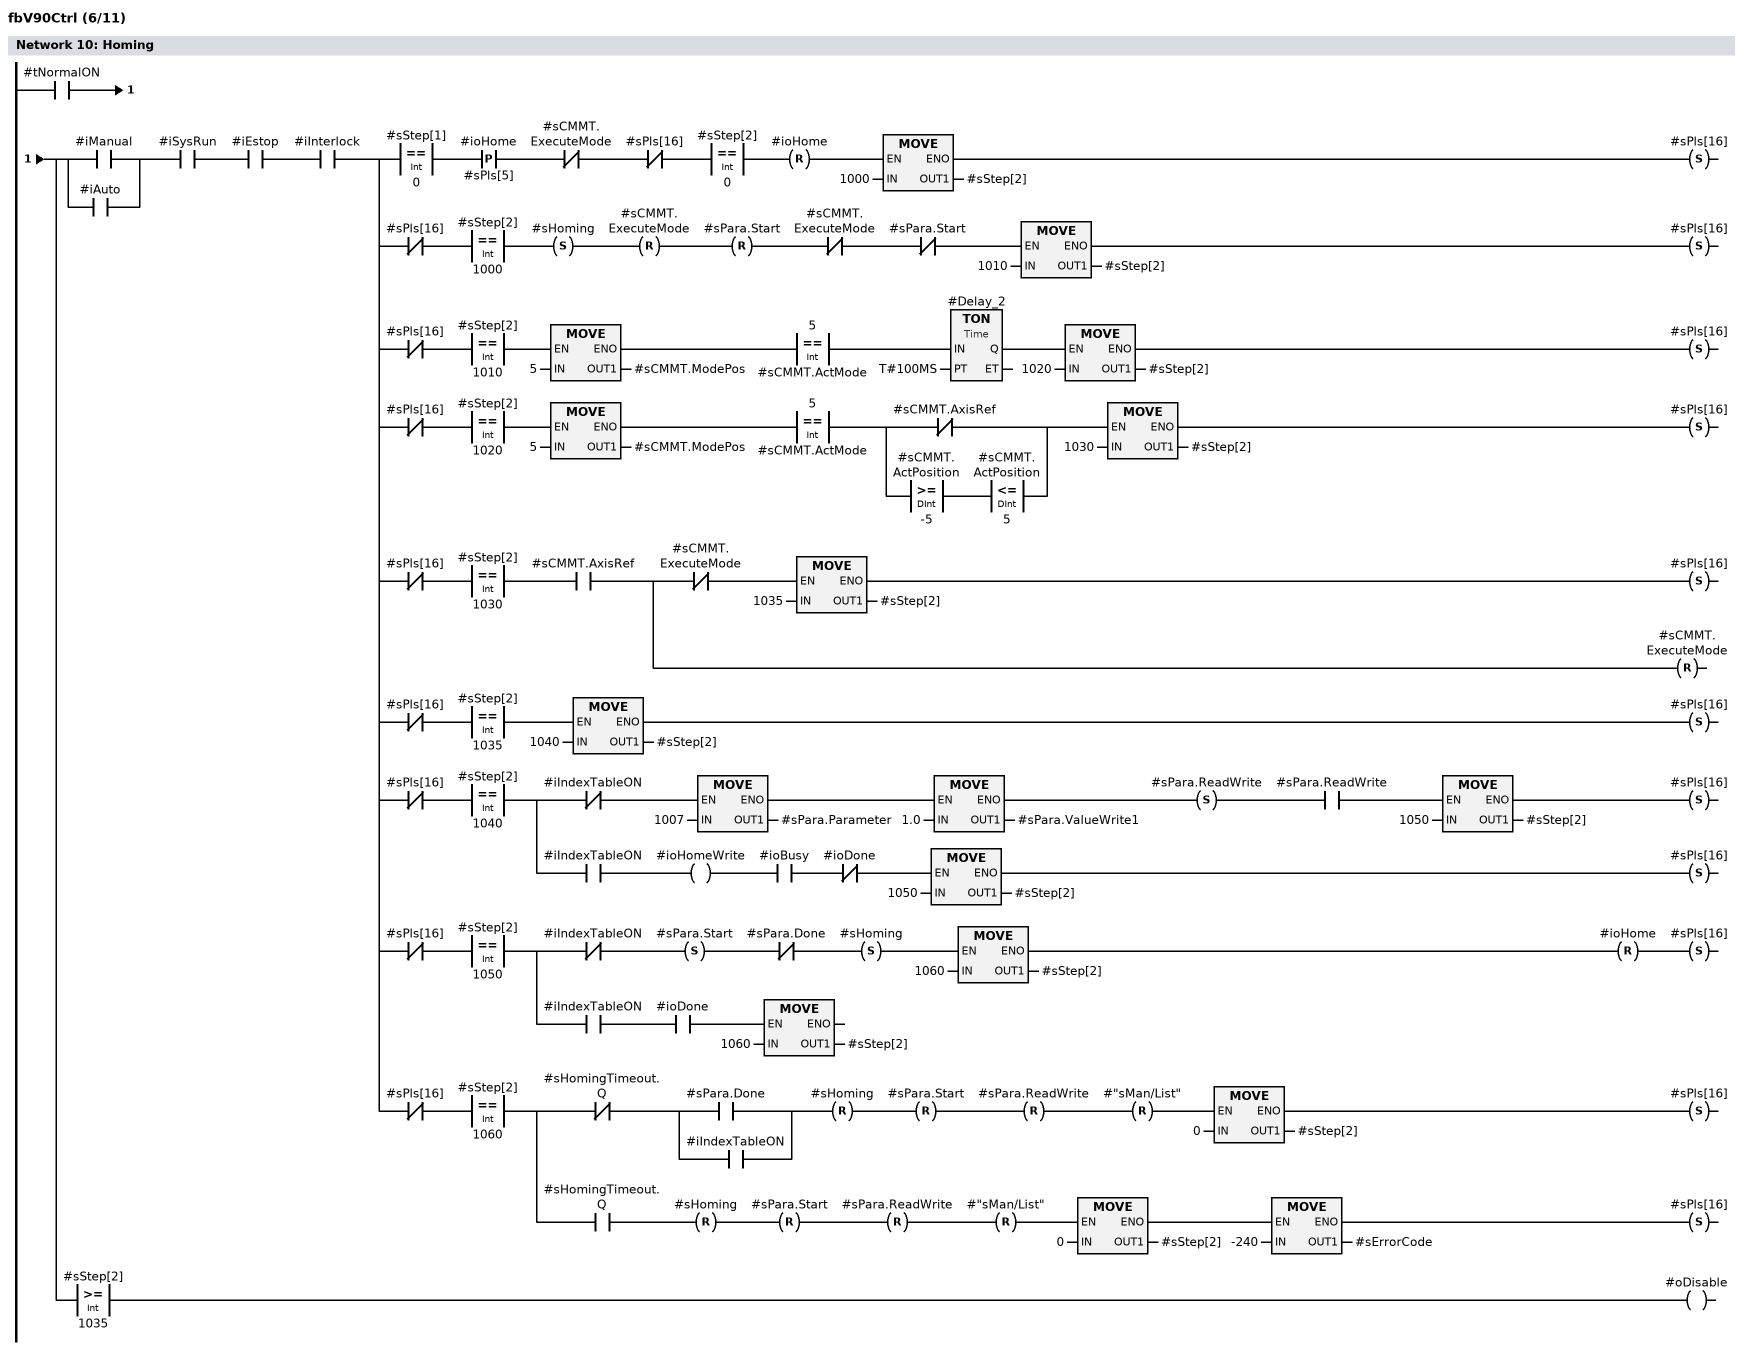
   RUNG wire#powerrail
      Contact( #tNormalON )
      wire#w1
      Contact( #iManual )
      wire#w2
      Contact( #iSysRun )
      Contact( #iEstop )
      Contact( #iInterlock )
      wire#w3
      { S7_Templates := "SrcType := Int" } EQ_Contact(in1 := #sStep[1], in2 := 0)
      P_Contact(operand := #ioHome, bit := #sPls[5])
      I_Contact( #sCMMT.ExecuteMode )
      I_Contact( #sPls[16] )
      { S7_Templates := "SrcType := Int" } EQ_Contact(in1 := #sStep[2], in2 := 0)
      R_Coil( #ioHome )
      Move(in := 1000, out1 => #sStep[2])
      S_Coil( #sPls[16] )
   END_RUNG
   RUNG wire#w1
      Contact( #iAuto )
   END_RUNG wire#w2
   RUNG wire#w3
      I_Contact( #sPls[16] )
      { S7_Templates := "SrcType := Int" } EQ_Contact(in1 := #sStep[2], in2 := 1000)
      S_Coil( #sHoming )
      R_Coil( #sCMMT.ExecuteMode )
      R_Coil( #sPara.Start )
      I_Contact( #sCMMT.ExecuteMode )
      I_Contact( #sPara.Start )
      Move(in := 1010, out1 => #sStep[2])
      S_Coil( #sPls[16] )
   END_RUNG
   RUNG wire#w3
      I_Contact( #sPls[16] )
      { S7_Templates := "SrcType := Int" } EQ_Contact(in1 := #sStep[2], in2 := 1010)
      Move(in := 5, out1 => #sCMMT.ModePos)
      { S7_Templates := "SrcType := Int" } EQ_Contact(in1 := 5, in2 := #sCMMT.ActMode)
      { S7_Templates := "time_type := Time" } #Delay_2.TON(pt := T#100MS, et =>)
      Move(in := 1020, out1 => #sStep[2])
      S_Coil( #sPls[16] )
   END_RUNG
   RUNG wire#w3
      I_Contact( #sPls[16] )
      { S7_Templates := "SrcType := Int" } EQ_Contact(in1 := #sStep[2], in2 := 1020)
      Move(in := 5, out1 => #sCMMT.ModePos)
      { S7_Templates := "SrcType := Int" } EQ_Contact(in1 := 5, in2 := #sCMMT.ActMode)
      wire#w4
      I_Contact( #sCMMT.AxisRef )
      wire#w5
      Move(in := 1030, out1 => #sStep[2])
      S_Coil( #sPls[16] )
   END_RUNG
   RUNG wire#w4
      { S7_Templates := "SrcType := DInt" } GE_Contact(in1 := #sCMMT.ActPosition, in2 := -5)
      { S7_Templates := "SrcType := DInt" } LE_Contact(in1 := #sCMMT.ActPosition, in2 := 5)
   END_RUNG wire#w5
   RUNG wire#w3
      I_Contact( #sPls[16] )
      { S7_Templates := "SrcType := Int" } EQ_Contact(in1 := #sStep[2], in2 := 1030)
      Contact( #sCMMT.AxisRef )
      wire#w6
      I_Contact( #sCMMT.ExecuteMode )
      Move(in := 1035, out1 => #sStep[2])
      S_Coil( #sPls[16] )
   END_RUNG
   RUNG wire#w6
      R_Coil( #sCMMT.ExecuteMode )
   END_RUNG
   RUNG wire#w3
      I_Contact( #sPls[16] )
      { S7_Templates := "SrcType := Int" } EQ_Contact(in1 := #sStep[2], in2 := 1035)
      Move(in := 1040, out1 => #sStep[2])
      S_Coil( #sPls[16] )
   END_RUNG
   RUNG wire#w3
      I_Contact( #sPls[16] )
      { S7_Templates := "SrcType := Int" } EQ_Contact(in1 := #sStep[2], in2 := 1040)
      wire#w7
      I_Contact( #iIndexTableON )
      Move(in := 1007, out1 => #sPara.Parameter)
      Move(in := 1.0, out1 => #sPara.ValueWrite1)
      S_Coil( #sPara.ReadWrite )
      Contact( #sPara.ReadWrite )
      Move(in := 1050, out1 => #sStep[2])
      S_Coil( #sPls[16] )
   END_RUNG
   RUNG wire#w7
      Contact( #iIndexTableON )
      Coil( #ioHomeWrite )
      Contact( #ioBusy )
      I_Contact( #ioDone )
      Move(in := 1050, out1 => #sStep[2])
      S_Coil( #sPls[16] )
   END_RUNG
   RUNG wire#w3
      I_Contact( #sPls[16] )
      { S7_Templates := "SrcType := Int" } EQ_Contact(in1 := #sStep[2], in2 := 1050)
      wire#w8
      I_Contact( #iIndexTableON )
      S_Coil( #sPara.Start )
      I_Contact( #sPara.Done )
      S_Coil( #sHoming )
      Move(in := 1060, out1 => #sStep[2])
      R_Coil( #ioHome )
      S_Coil( #sPls[16] )
   END_RUNG
   RUNG wire#w8
      Contact( #iIndexTableON )
      Contact( #ioDone )
      Move(in := 1060, out1 => #sStep[2])
   END_RUNG
   RUNG wire#w3
      I_Contact( #sPls[16] )
      { S7_Templates := "SrcType := Int" } EQ_Contact(in1 := #sStep[2], in2 := 1060)
      wire#w9
      I_Contact( #sHomingTimeout.Q )
      wire#w10
      Contact( #sPara.Done )
      wire#w11
      R_Coil( #sHoming )
      R_Coil( #sPara.Start )
      R_Coil( #sPara.ReadWrite )
      R_Coil( #"sMan/List" )
      Move(in := 0, out1 => #sStep[2])
      S_Coil( #sPls[16] )
   END_RUNG
   RUNG wire#w10
      Contact( #iIndexTableON )
   END_RUNG wire#w11
   RUNG wire#w9
      Contact( #sHomingTimeout.Q )
      R_Coil( #sHoming )
      R_Coil( #sPara.Start )
      R_Coil( #sPara.ReadWrite )
      R_Coil( #"sMan/List" )
      Move(in := 0, out1 => #sStep[2])
      Move(in := -240, out1 => #sErrorCode)
      S_Coil( #sPls[16] )
   END_RUNG
   RUNG wire#w1
      { S7_Templates := "SrcType := Int" } GE_Contact(in1 := #sStep[2], in2 := 1035)
      Coil( #oDisable )
   END_RUNG
   // the same network as SCL:
   #_w1 := #tNormalON AND (#iManual OR #iAuto) AND #iSysRun AND #iEstop AND #iInterlock;
   #_w2 := #_w1 AND (#sStep[1] = 0) AND #ioHome AND NOT #sPls[5];   // rising edge of #ioHome
   #sPls[5] := #ioHome;
   IF #_w2 AND NOT #sCMMT.ExecuteMode AND NOT #sPls[16] AND (#sStep[2] = 0) THEN #ioHome := FALSE; END_IF;
   #_w3 := #_w2 AND NOT #sCMMT.ExecuteMode AND NOT #sPls[16] AND (#sStep[2] = 0);
   IF #_w3 THEN
       #sStep[2] := 1000;
       #sPls[16] := TRUE;
   END_IF;
   #_w4 := #_w1 AND NOT #sPls[16] AND (#sStep[2] = 1000);
   IF #_w4 THEN
       #sHoming := TRUE;
       #sCMMT.ExecuteMode := FALSE;
       #sPara.Start := FALSE;
   END_IF;
   IF #_w4 AND NOT #sCMMT.ExecuteMode AND NOT #sPara.Start THEN
       #sStep[2] := 1010;
       #sPls[16] := TRUE;
   END_IF;
   #_w5 := #_w1 AND NOT #sPls[16] AND (#sStep[2] = 1010);
   IF #_w5 THEN #sCMMT.ModePos := 5; END_IF;
   #Delay_2(IN := #_w5 AND (5 = #sCMMT.ActMode), PT := T#100MS);   // TON
   IF #Delay_2.Q THEN
       #sStep[2] := 1020;
       #sPls[16] := TRUE;
   END_IF;
   #_w6 := #_w1 AND NOT #sPls[16] AND (#sStep[2] = 1020);
   IF #_w6 THEN #sCMMT.ModePos := 5; END_IF;
   IF #_w6 AND (5 = #sCMMT.ActMode) AND (NOT #sCMMT.AxisRef OR ((#sCMMT.ActPosition >= (-5)) AND (#sCMMT.ActPosition <= 5))) THEN
       #sStep[2] := 1030;
       #sPls[16] := TRUE;
   END_IF;
   #_w7 := #_w1 AND NOT #sPls[16] AND (#sStep[2] = 1030) AND #sCMMT.AxisRef;
   IF #_w7 AND NOT #sCMMT.ExecuteMode THEN
       #sStep[2] := 1035;
       #sPls[16] := TRUE;
   END_IF;
   IF #_w7 THEN #sCMMT.ExecuteMode := FALSE; END_IF;
   #_w8 := #_w1 AND NOT #sPls[16] AND (#sStep[2] = 1035);
   IF #_w8 THEN
       #sStep[2] := 1040;
       #sPls[16] := TRUE;
   END_IF;
   #_w9 := #_w1 AND NOT #sPls[16] AND (#sStep[2] = 1040);
   #_w10 := #_w9 AND NOT #iIndexTableON;
   IF #_w10 THEN
       #sPara.Parameter := 1007;
       #sPara.ValueWrite1 := 1.0;
       #sPara.ReadWrite := TRUE;
   END_IF;
   IF #_w10 AND #sPara.ReadWrite THEN
       #sStep[2] := 1050;
       #sPls[16] := TRUE;
   END_IF;
   #ioHomeWrite := #_w9 AND #iIndexTableON;
   IF #ioHomeWrite AND #ioBusy AND NOT #ioDone THEN
       #sStep[2] := 1050;
       #sPls[16] := TRUE;
   END_IF;
   #_w11 := #_w1 AND NOT #sPls[16] AND (#sStep[2] = 1050);
   #_w12 := #_w11 AND NOT #iIndexTableON;
   IF #_w12 THEN #sPara.Start := TRUE; END_IF;
   IF #_w12 AND NOT #sPara.Done THEN
       #sHoming := TRUE;
       #sStep[2] := 1060;
       #ioHome := FALSE;
       #sPls[16] := TRUE;
   END_IF;
   IF #_w11 AND #iIndexTableON AND #ioDone THEN #sStep[2] := 1060; END_IF;
   #_w13 := #_w1 AND NOT #sPls[16] AND (#sStep[2] = 1060);
   IF #_w13 AND NOT #sHomingTimeout.Q AND (#sPara.Done OR #iIndexTableON) THEN
       #sHoming := FALSE;
       #sPara.Start := FALSE;
       #sPara.ReadWrite := FALSE;
       #"sMan/List" := FALSE;
       #sStep[2] := 0;
       #sPls[16] := TRUE;
   END_IF;
   IF #_w13 AND #sHomingTimeout.Q THEN
       #sHoming := FALSE;
       #sPara.Start := FALSE;
       #sPara.ReadWrite := FALSE;
       #"sMan/List" := FALSE;
       #sStep[2] := 0;
       #sErrorCode := -240;
       #sPls[16] := TRUE;
   END_IF;
   #oDisable := #tNormalON AND (#sStep[2] >= 1035);
END_REGION

REGION Network 11: HomingTimeout
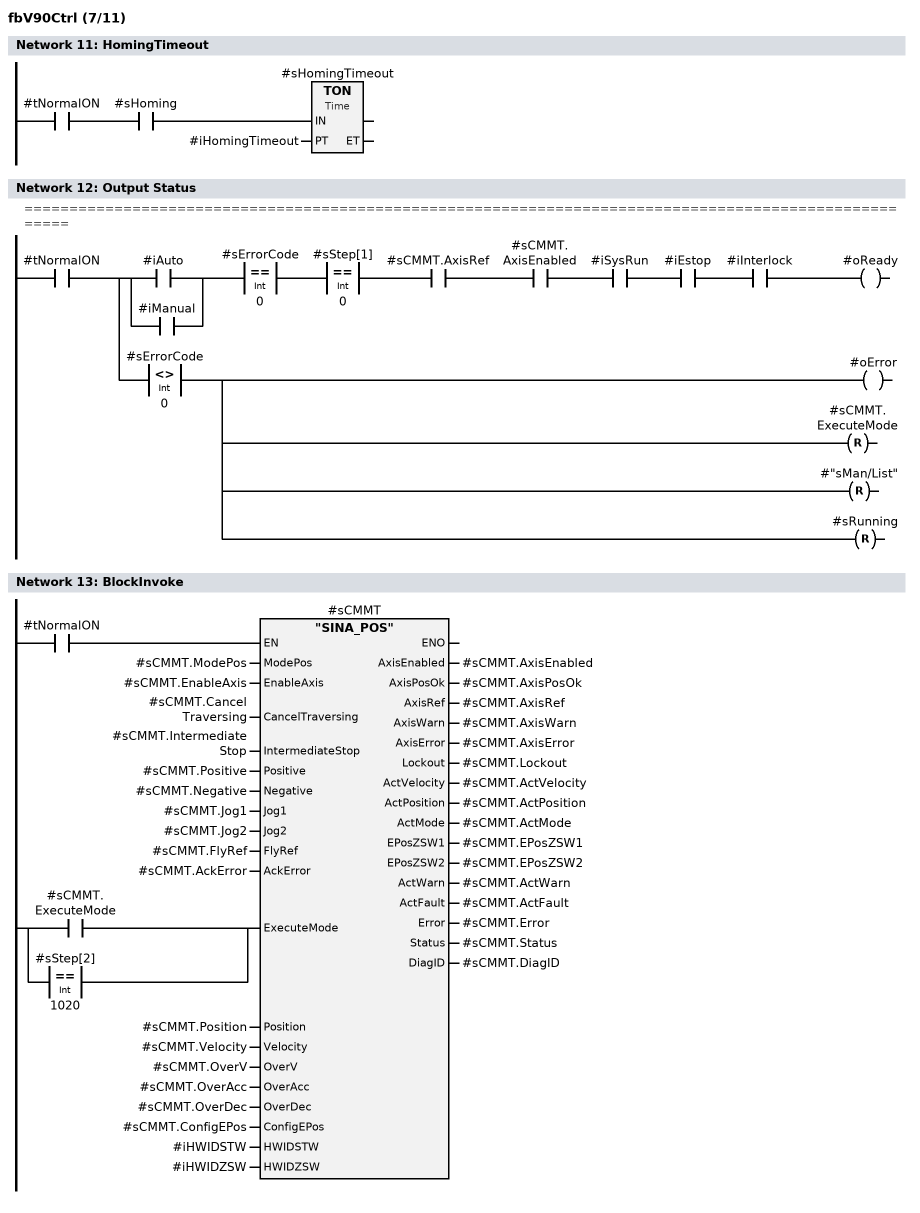
   RUNG wire#powerrail
      Contact( #tNormalON )
      Contact( #sHoming )
      { S7_Templates := "time_type := Time" } #sHomingTimeout.TON(pt := #iHomingTimeout, et =>)
   END_RUNG
   // the same network as SCL:
   #sHomingTimeout(IN := #tNormalON AND #sHoming, PT := #iHomingTimeout);   // TON
END_REGION

REGION Network 12: Output Status
   // ======================================================================================================
   RUNG wire#powerrail
      Contact( #tNormalON )
      wire#w1
      Contact( #iAuto )
      wire#w2
      { S7_Templates := "SrcType := Int" } EQ_Contact(in1 := #sErrorCode, in2 := 0)
      { S7_Templates := "SrcType := Int" } EQ_Contact(in1 := #sStep[1], in2 := 0)
      Contact( #sCMMT.AxisRef )
      Contact( #sCMMT.AxisEnabled )
      Contact( #iSysRun )
      Contact( #iEstop )
      Contact( #iInterlock )
      Coil( #oReady )
   END_RUNG
   RUNG wire#w1
      Contact( #iManual )
   END_RUNG wire#w2
   RUNG wire#w1
      { S7_Templates := "SrcType := Int" } NE_Contact(in1 := #sErrorCode, in2 := 0)
      wire#w3
      Coil( #oError )
   END_RUNG
   RUNG wire#w3
      R_Coil( #sCMMT.ExecuteMode )
   END_RUNG
   RUNG wire#w3
      R_Coil( #"sMan/List" )
   END_RUNG
   RUNG wire#w3
      R_Coil( #sRunning )
   END_RUNG
   // the same network as SCL:
   #oReady := #tNormalON AND (#iAuto OR #iManual) AND (#sErrorCode = 0) AND (#sStep[1] = 0) AND #sCMMT.AxisRef AND #sCMMT.AxisEnabled AND #iSysRun AND #iEstop AND #iInterlock;
   #oError := #tNormalON AND (#sErrorCode <> 0);
   IF #oError THEN
       #sCMMT.ExecuteMode := FALSE;
       #"sMan/List" := FALSE;
       #sRunning := FALSE;
   END_IF;
END_REGION

REGION Network 13: BlockInvoke
   RUNG wire#powerrail
      Contact( #tNormalON )
      #sCMMT(ExecuteMode := wire#w1, ModePos := #sCMMT.ModePos, EnableAxis := #sCMMT.EnableAxis, CancelTraversing := #sCMMT.CancelTraversing, IntermediateStop := #sCMMT.IntermediateStop, Positive := #sCMMT.Positive, Negative := #sCMMT.Negative, Jog1 := #sCMMT.Jog1, Jog2 := #sCMMT.Jog2, FlyRef := #sCMMT.FlyRef, AckError := #sCMMT.AckError, Position := #sCMMT.Position, Velocity := #sCMMT.Velocity, OverV := #sCMMT.OverV, OverAcc := #sCMMT.OverAcc, OverDec := #sCMMT.OverDec, ConfigEPos := #sCMMT.ConfigEPos, HWIDSTW := #iHWIDSTW, HWIDZSW := #iHWIDZSW, AxisEnabled => #sCMMT.AxisEnabled, AxisPosOk => #sCMMT.AxisPosOk, AxisRef => #sCMMT.AxisRef, AxisWarn => #sCMMT.AxisWarn, AxisError => #sCMMT.AxisError, Lockout => #sCMMT.Lockout, ActVelocity => #sCMMT.ActVelocity, ActPosition => #sCMMT.ActPosition, ActMode => #sCMMT.ActMode, EPosZSW1 => #sCMMT.EPosZSW1, EPosZSW2 => #sCMMT.EPosZSW2, ActWarn => #sCMMT.ActWarn, ActFault => #sCMMT.ActFault, Error => #sCMMT.Error, Status => #sCMMT.Status, DiagID => #sCMMT.DiagID)
   END_RUNG
   RUNG wire#powerrail
      Contact( #sCMMT.ExecuteMode )
   END_RUNG wire#w1
   RUNG wire#powerrail
      { S7_Templates := "SrcType := Int" } EQ_Contact(in1 := #sStep[2], in2 := 1020)
   END_RUNG wire#w1
   // the same network as SCL:
   IF #tNormalON THEN
       #sCMMT(ModePos := #sCMMT.ModePos,   // "SINA_POS"
              EnableAxis := #sCMMT.EnableAxis,
              CancelTraversing := #sCMMT.CancelTraversing,
              IntermediateStop := #sCMMT.IntermediateStop,
              Positive := #sCMMT.Positive,
              Negative := #sCMMT.Negative,
              Jog1 := #sCMMT.Jog1,
              Jog2 := #sCMMT.Jog2,
              FlyRef := #sCMMT.FlyRef,
              AckError := #sCMMT.AckError,
              ExecuteMode := #sCMMT.ExecuteMode OR (#sStep[2] = 1020),
              Position := #sCMMT.Position,
              Velocity := #sCMMT.Velocity,
              OverV := #sCMMT.OverV,
              OverAcc := #sCMMT.OverAcc,
              OverDec := #sCMMT.OverDec,
              ConfigEPos := #sCMMT.ConfigEPos,
              HWIDSTW := #iHWIDSTW,
              HWIDZSW := #iHWIDZSW,
              AxisEnabled => #sCMMT.AxisEnabled,
              AxisPosOk => #sCMMT.AxisPosOk,
              AxisRef => #sCMMT.AxisRef,
              AxisWarn => #sCMMT.AxisWarn,
              AxisError => #sCMMT.AxisError,
              Lockout => #sCMMT.Lockout,
              ActVelocity => #sCMMT.ActVelocity,
              ActPosition => #sCMMT.ActPosition,
              ActMode => #sCMMT.ActMode,
              EPosZSW1 => #sCMMT.EPosZSW1,
              EPosZSW2 => #sCMMT.EPosZSW2,
              ActWarn => #sCMMT.ActWarn,
              ActFault => #sCMMT.ActFault,
              Error => #sCMMT.Error,
              Status => #sCMMT.Status,
              DiagID => #sCMMT.DiagID);
   END_IF;
END_REGION

REGION Network 14: BlockInvoke
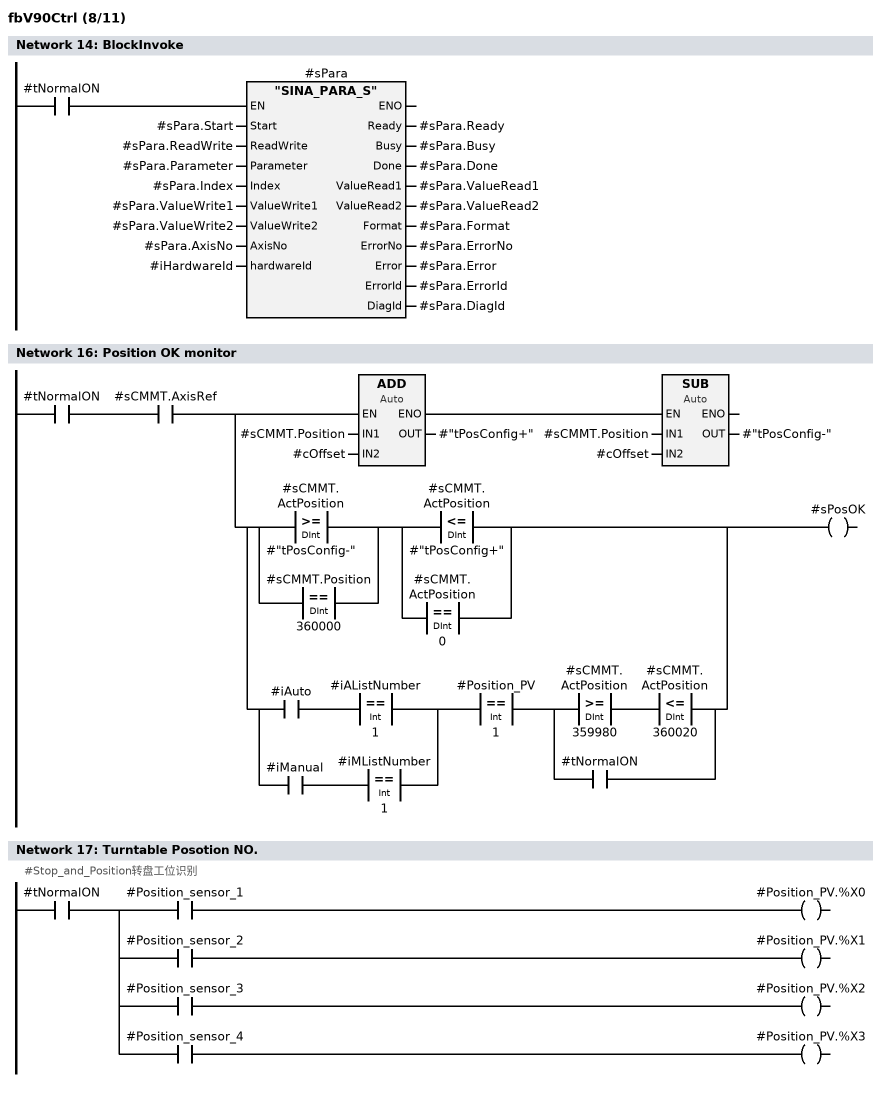
   RUNG wire#powerrail
      Contact( #tNormalON )
      #sPara(Start := #sPara.Start, ReadWrite := #sPara.ReadWrite, Parameter := #sPara.Parameter, Index := #sPara.Index, ValueWrite1 := #sPara.ValueWrite1, ValueWrite2 := #sPara.ValueWrite2, AxisNo := #sPara.AxisNo, hardwareId := #iHardwareId, Ready => #sPara.Ready, Busy => #sPara.Busy, Done => #sPara.Done, ValueRead1 => #sPara.ValueRead1, ValueRead2 => #sPara.ValueRead2, Format => #sPara.Format, ErrorNo => #sPara.ErrorNo, Error => #sPara.Error, ErrorId => #sPara.ErrorId, DiagId => #sPara.DiagId)
   END_RUNG
   // the same network as SCL:
   IF #tNormalON THEN
       #sPara(Start := #sPara.Start,   // "SINA_PARA_S"
              ReadWrite := #sPara.ReadWrite,
              Parameter := #sPara.Parameter,
              Index := #sPara.Index,
              ValueWrite1 := #sPara.ValueWrite1,
              ValueWrite2 := #sPara.ValueWrite2,
              AxisNo := #sPara.AxisNo,
              hardwareId := #iHardwareId,
              Ready => #sPara.Ready,
              Busy => #sPara.Busy,
              Done => #sPara.Done,
              ValueRead1 => #sPara.ValueRead1,
              ValueRead2 => #sPara.ValueRead2,
              Format => #sPara.Format,
              ErrorNo => #sPara.ErrorNo,
              Error => #sPara.Error,
              ErrorId => #sPara.ErrorId,
              DiagId => #sPara.DiagId);
   END_IF;
END_REGION

REGION Network 16: Position OK monitor
   RUNG wire#powerrail
      Contact( #tNormalON )
      Contact( #sCMMT.AxisRef )
      wire#w1
      Add(in1 := #sCMMT.Position, in2 := #cOffset, out => #"tPosConfig+")
      Sub(in1 := #sCMMT.Position, in2 := #cOffset, out => #"tPosConfig-")
   END_RUNG
   RUNG wire#w1
      { S7_Templates := "SrcType := DInt" } GE_Contact(in1 := #sCMMT.ActPosition, in2 := #"tPosConfig-")
      wire#w2
      { S7_Templates := "SrcType := DInt" } LE_Contact(in1 := #sCMMT.ActPosition, in2 := #"tPosConfig+")
      wire#w3
      Coil( #sPosOK )
   END_RUNG
   RUNG wire#w1
      { S7_Templates := "SrcType := DInt" } EQ_Contact(in1 := #sCMMT.Position, in2 := 360000)
   END_RUNG wire#w2
   RUNG wire#w2
      { S7_Templates := "SrcType := DInt" } EQ_Contact(in1 := #sCMMT.ActPosition, in2 := 0)
   END_RUNG wire#w3
   RUNG wire#w1
      Contact( #iAuto )
      { S7_Templates := "SrcType := Int" } EQ_Contact(in1 := #iAListNumber, in2 := 1)
      wire#w4
      { S7_Templates := "SrcType := Int" } EQ_Contact(in1 := #Position_PV, in2 := 1)
      wire#w5
      { S7_Templates := "SrcType := DInt" } GE_Contact(in1 := #sCMMT.ActPosition, in2 := 359980)
      { S7_Templates := "SrcType := DInt" } LE_Contact(in1 := #sCMMT.ActPosition, in2 := 360020)
   END_RUNG wire#w3
   RUNG wire#w1
      Contact( #iManual )
      { S7_Templates := "SrcType := Int" } EQ_Contact(in1 := #iMListNumber, in2 := 1)
   END_RUNG wire#w4
   RUNG wire#w5
      Contact( #tNormalON )
   END_RUNG wire#w3
   // the same network as SCL:
   #_w1 := #tNormalON AND #sCMMT.AxisRef;
   IF #_w1 THEN
       #"tPosConfig+" := #sCMMT.Position + #cOffset;
       #"tPosConfig-" := #sCMMT.Position - #cOffset;
   END_IF;
   #sPosOK := #_w1 AND ((((#sCMMT.ActPosition >= #"tPosConfig-") OR (#sCMMT.Position = 360000)) AND ((#sCMMT.ActPosition <= #"tPosConfig+") OR (#sCMMT.ActPosition = 0))) OR (((#iAuto AND (#iAListNumber = 1)) OR (#iManual AND (#iMListNumber = 1))) AND (#Position_PV = 1) AND (((#sCMMT.ActPosition >= 359980) AND (#sCMMT.ActPosition <= 360020)) OR #tNormalON)));
END_REGION

REGION Network 17: Turntable Posotion NO.
   // #Stop_and_Position转盘工位识别
   RUNG wire#powerrail
      Contact( #tNormalON )
      wire#w1
      Contact( #Position_sensor_1 )
      Coil( #Position_PV.%X0 )
   END_RUNG
   RUNG wire#w1
      Contact( #Position_sensor_2 )
      Coil( #Position_PV.%X1 )
   END_RUNG
   RUNG wire#w1
      Contact( #Position_sensor_3 )
      Coil( #Position_PV.%X2 )
   END_RUNG
   RUNG wire#w1
      Contact( #Position_sensor_4 )
      Coil( #Position_PV.%X3 )
   END_RUNG
   // the same network as SCL:
   #Position_PV.%X0 := #tNormalON AND #Position_sensor_1;
   #Position_PV.%X1 := #tNormalON AND #Position_sensor_2;
   #Position_PV.%X2 := #tNormalON AND #Position_sensor_3;
   #Position_PV.%X3 := #tNormalON AND #Position_sensor_4;
END_REGION

REGION Network 18: 根据识别号 转换位位置号 / Convert the bit position number from the identification number
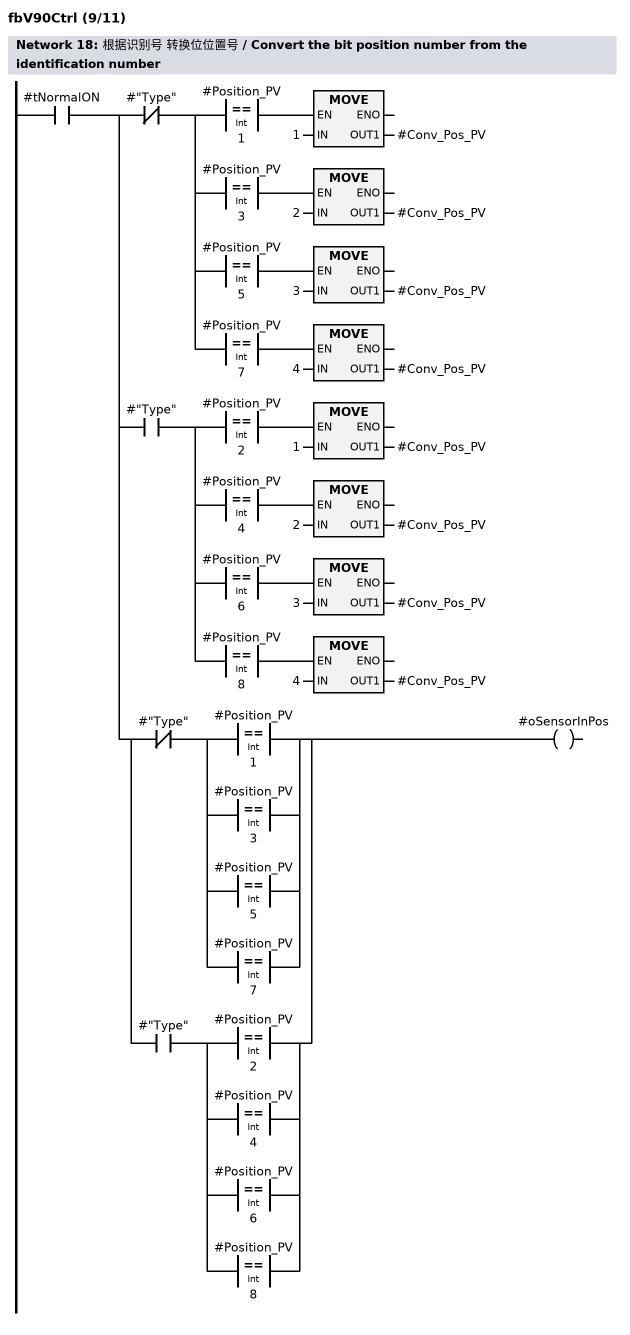
   RUNG wire#powerrail
      Contact( #tNormalON )
      wire#w1
      I_Contact( #"Type" )
      wire#w2
      { S7_Templates := "SrcType := Int" } EQ_Contact(in1 := #Position_PV, in2 := 1)
      Move(in := 1, out1 => #Conv_Pos_PV)
   END_RUNG
   RUNG wire#w2
      { S7_Templates := "SrcType := Int" } EQ_Contact(in1 := #Position_PV, in2 := 3)
      Move(in := 2, out1 => #Conv_Pos_PV)
   END_RUNG
   RUNG wire#w2
      { S7_Templates := "SrcType := Int" } EQ_Contact(in1 := #Position_PV, in2 := 5)
      Move(in := 3, out1 => #Conv_Pos_PV)
   END_RUNG
   RUNG wire#w2
      { S7_Templates := "SrcType := Int" } EQ_Contact(in1 := #Position_PV, in2 := 7)
      Move(in := 4, out1 => #Conv_Pos_PV)
   END_RUNG
   RUNG wire#w1
      Contact( #"Type" )
      wire#w3
      { S7_Templates := "SrcType := Int" } EQ_Contact(in1 := #Position_PV, in2 := 2)
      Move(in := 1, out1 => #Conv_Pos_PV)
   END_RUNG
   RUNG wire#w3
      { S7_Templates := "SrcType := Int" } EQ_Contact(in1 := #Position_PV, in2 := 4)
      Move(in := 2, out1 => #Conv_Pos_PV)
   END_RUNG
   RUNG wire#w3
      { S7_Templates := "SrcType := Int" } EQ_Contact(in1 := #Position_PV, in2 := 6)
      Move(in := 3, out1 => #Conv_Pos_PV)
   END_RUNG
   RUNG wire#w3
      { S7_Templates := "SrcType := Int" } EQ_Contact(in1 := #Position_PV, in2 := 8)
      Move(in := 4, out1 => #Conv_Pos_PV)
   END_RUNG
   RUNG wire#w1
      I_Contact( #"Type" )
      wire#w4
      { S7_Templates := "SrcType := Int" } EQ_Contact(in1 := #Position_PV, in2 := 1)
      wire#w5
      Coil( #oSensorInPos )
   END_RUNG
   RUNG wire#w4
      { S7_Templates := "SrcType := Int" } EQ_Contact(in1 := #Position_PV, in2 := 3)
   END_RUNG wire#w5
   RUNG wire#w4
      { S7_Templates := "SrcType := Int" } EQ_Contact(in1 := #Position_PV, in2 := 5)
   END_RUNG wire#w5
   RUNG wire#w4
      { S7_Templates := "SrcType := Int" } EQ_Contact(in1 := #Position_PV, in2 := 7)
   END_RUNG wire#w5
   RUNG wire#w1
      Contact( #"Type" )
      wire#w6
      { S7_Templates := "SrcType := Int" } EQ_Contact(in1 := #Position_PV, in2 := 2)
   END_RUNG wire#w5
   RUNG wire#w6
      { S7_Templates := "SrcType := Int" } EQ_Contact(in1 := #Position_PV, in2 := 4)
   END_RUNG wire#w5
   RUNG wire#w6
      { S7_Templates := "SrcType := Int" } EQ_Contact(in1 := #Position_PV, in2 := 6)
   END_RUNG wire#w5
   RUNG wire#w6
      { S7_Templates := "SrcType := Int" } EQ_Contact(in1 := #Position_PV, in2 := 8)
   END_RUNG wire#w5
   // the same network as SCL:
   #_w1 := #tNormalON AND NOT #"Type";
   IF #_w1 AND (#Position_PV = 1) THEN #Conv_Pos_PV := 1; END_IF;
   IF #_w1 AND (#Position_PV = 3) THEN #Conv_Pos_PV := 2; END_IF;
   IF #_w1 AND (#Position_PV = 5) THEN #Conv_Pos_PV := 3; END_IF;
   IF #_w1 AND (#Position_PV = 7) THEN #Conv_Pos_PV := 4; END_IF;
   #_w2 := #tNormalON AND #"Type";
   IF #_w2 AND (#Position_PV = 2) THEN #Conv_Pos_PV := 1; END_IF;
   IF #_w2 AND (#Position_PV = 4) THEN #Conv_Pos_PV := 2; END_IF;
   IF #_w2 AND (#Position_PV = 6) THEN #Conv_Pos_PV := 3; END_IF;
   IF #_w2 AND (#Position_PV = 8) THEN #Conv_Pos_PV := 4; END_IF;
   #oSensorInPos := #tNormalON AND ((NOT #"Type" AND ((#Position_PV = 1) OR (#Position_PV = 3) OR (#Position_PV = 5) OR (#Position_PV = 7))) OR (#"Type" AND ((#Position_PV = 2) OR (#Position_PV = 4) OR (#Position_PV = 6) OR (#Position_PV = 8))));
END_REGION

REGION Network 19: Pos OK/Pos done
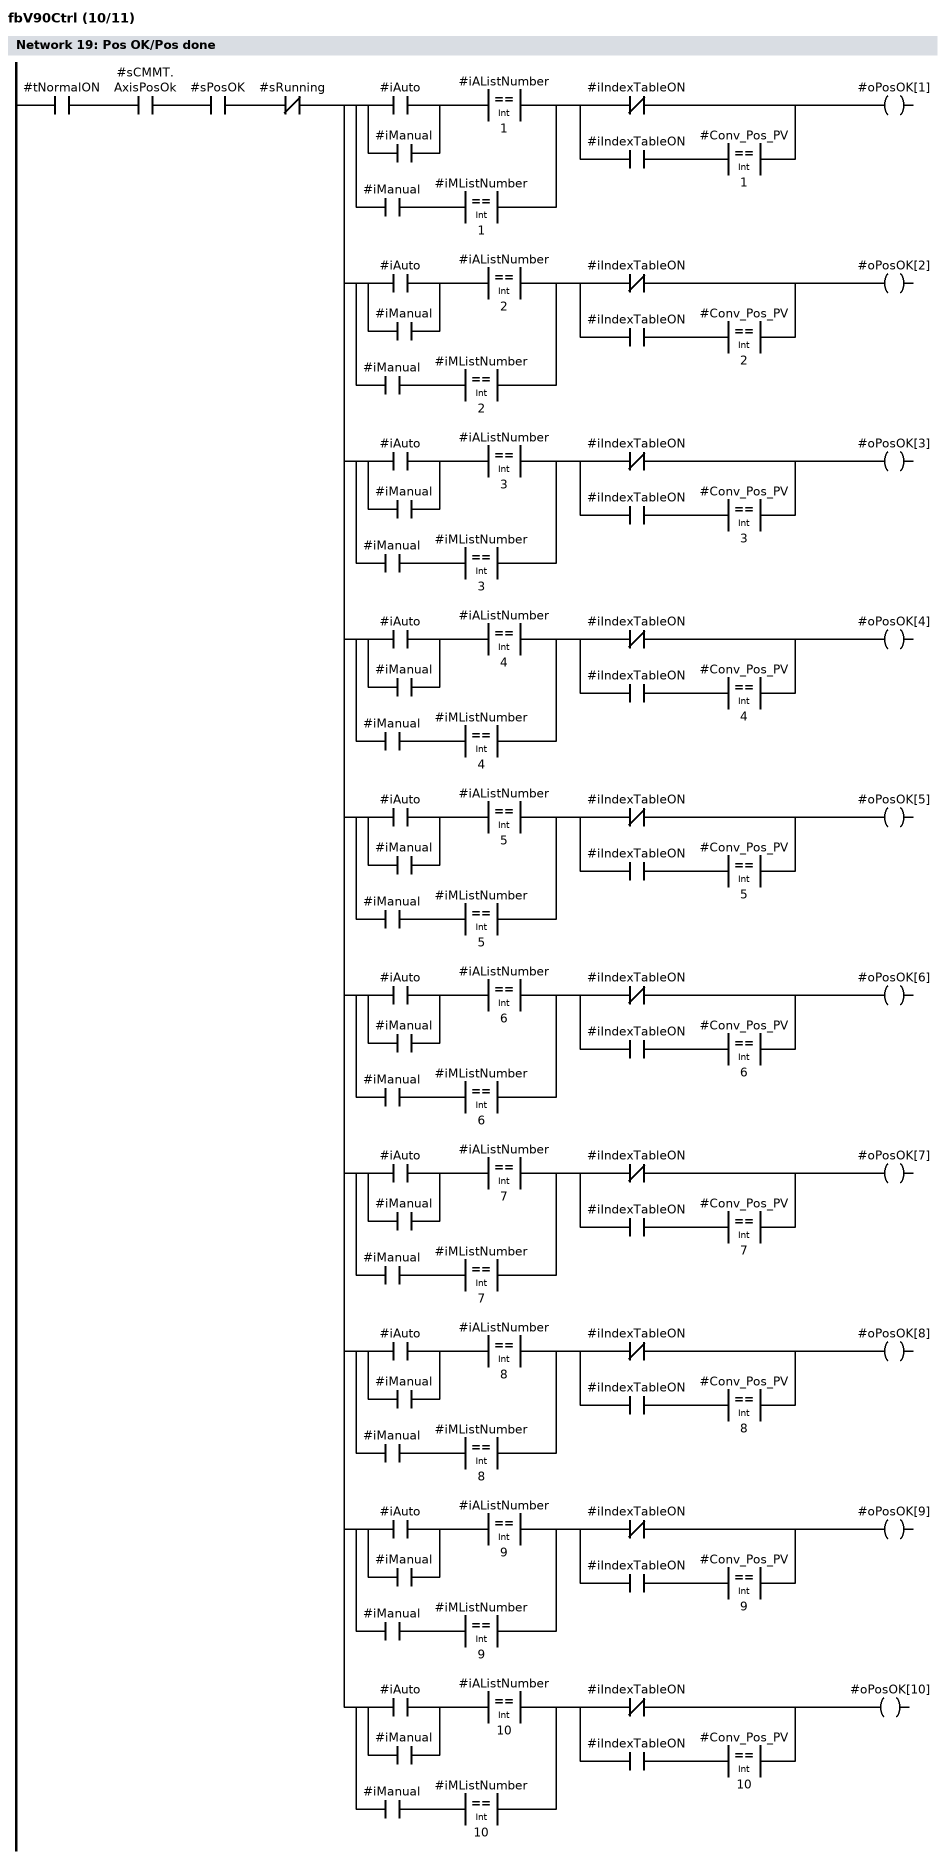
   RUNG wire#powerrail
      Contact( #tNormalON )
      Contact( #sCMMT.AxisPosOk )
      Contact( #sPosOK )
      I_Contact( #sRunning )
      wire#w1
      Contact( #iAuto )
      wire#w2
      { S7_Templates := "SrcType := Int" } EQ_Contact(in1 := #iAListNumber, in2 := 1)
      wire#w3
      I_Contact( #iIndexTableON )
      wire#w4
      Coil( #oPosOK[1] )
   END_RUNG
   RUNG wire#w1
      Contact( #iManual )
   END_RUNG wire#w2
   RUNG wire#w1
      Contact( #iManual )
      { S7_Templates := "SrcType := Int" } EQ_Contact(in1 := #iMListNumber, in2 := 1)
   END_RUNG wire#w3
   RUNG wire#w3
      Contact( #iIndexTableON )
      { S7_Templates := "SrcType := Int" } EQ_Contact(in1 := #Conv_Pos_PV, in2 := 1)
   END_RUNG wire#w4
   RUNG wire#w1
      Contact( #iAuto )
      wire#w5
      { S7_Templates := "SrcType := Int" } EQ_Contact(in1 := #iAListNumber, in2 := 2)
      wire#w6
      I_Contact( #iIndexTableON )
      wire#w7
      Coil( #oPosOK[2] )
   END_RUNG
   RUNG wire#w1
      Contact( #iManual )
   END_RUNG wire#w5
   RUNG wire#w1
      Contact( #iManual )
      { S7_Templates := "SrcType := Int" } EQ_Contact(in1 := #iMListNumber, in2 := 2)
   END_RUNG wire#w6
   RUNG wire#w6
      Contact( #iIndexTableON )
      { S7_Templates := "SrcType := Int" } EQ_Contact(in1 := #Conv_Pos_PV, in2 := 2)
   END_RUNG wire#w7
   RUNG wire#w1
      Contact( #iAuto )
      wire#w8
      { S7_Templates := "SrcType := Int" } EQ_Contact(in1 := #iAListNumber, in2 := 3)
      wire#w9
      I_Contact( #iIndexTableON )
      wire#w10
      Coil( #oPosOK[3] )
   END_RUNG
   RUNG wire#w1
      Contact( #iManual )
   END_RUNG wire#w8
   RUNG wire#w1
      Contact( #iManual )
      { S7_Templates := "SrcType := Int" } EQ_Contact(in1 := #iMListNumber, in2 := 3)
   END_RUNG wire#w9
   RUNG wire#w9
      Contact( #iIndexTableON )
      { S7_Templates := "SrcType := Int" } EQ_Contact(in1 := #Conv_Pos_PV, in2 := 3)
   END_RUNG wire#w10
   RUNG wire#w1
      Contact( #iAuto )
      wire#w11
      { S7_Templates := "SrcType := Int" } EQ_Contact(in1 := #iAListNumber, in2 := 4)
      wire#w12
      I_Contact( #iIndexTableON )
      wire#w13
      Coil( #oPosOK[4] )
   END_RUNG
   RUNG wire#w1
      Contact( #iManual )
   END_RUNG wire#w11
   RUNG wire#w1
      Contact( #iManual )
      { S7_Templates := "SrcType := Int" } EQ_Contact(in1 := #iMListNumber, in2 := 4)
   END_RUNG wire#w12
   RUNG wire#w12
      Contact( #iIndexTableON )
      { S7_Templates := "SrcType := Int" } EQ_Contact(in1 := #Conv_Pos_PV, in2 := 4)
   END_RUNG wire#w13
   RUNG wire#w1
      Contact( #iAuto )
      wire#w14
      { S7_Templates := "SrcType := Int" } EQ_Contact(in1 := #iAListNumber, in2 := 5)
      wire#w15
      I_Contact( #iIndexTableON )
      wire#w16
      Coil( #oPosOK[5] )
   END_RUNG
   RUNG wire#w1
      Contact( #iManual )
   END_RUNG wire#w14
   RUNG wire#w1
      Contact( #iManual )
      { S7_Templates := "SrcType := Int" } EQ_Contact(in1 := #iMListNumber, in2 := 5)
   END_RUNG wire#w15
   RUNG wire#w15
      Contact( #iIndexTableON )
      { S7_Templates := "SrcType := Int" } EQ_Contact(in1 := #Conv_Pos_PV, in2 := 5)
   END_RUNG wire#w16
   RUNG wire#w1
      Contact( #iAuto )
      wire#w17
      { S7_Templates := "SrcType := Int" } EQ_Contact(in1 := #iAListNumber, in2 := 6)
      wire#w18
      I_Contact( #iIndexTableON )
      wire#w19
      Coil( #oPosOK[6] )
   END_RUNG
   RUNG wire#w1
      Contact( #iManual )
   END_RUNG wire#w17
   RUNG wire#w1
      Contact( #iManual )
      { S7_Templates := "SrcType := Int" } EQ_Contact(in1 := #iMListNumber, in2 := 6)
   END_RUNG wire#w18
   RUNG wire#w18
      Contact( #iIndexTableON )
      { S7_Templates := "SrcType := Int" } EQ_Contact(in1 := #Conv_Pos_PV, in2 := 6)
   END_RUNG wire#w19
   RUNG wire#w1
      Contact( #iAuto )
      wire#w20
      { S7_Templates := "SrcType := Int" } EQ_Contact(in1 := #iAListNumber, in2 := 7)
      wire#w21
      I_Contact( #iIndexTableON )
      wire#w22
      Coil( #oPosOK[7] )
   END_RUNG
   RUNG wire#w1
      Contact( #iManual )
   END_RUNG wire#w20
   RUNG wire#w1
      Contact( #iManual )
      { S7_Templates := "SrcType := Int" } EQ_Contact(in1 := #iMListNumber, in2 := 7)
   END_RUNG wire#w21
   RUNG wire#w21
      Contact( #iIndexTableON )
      { S7_Templates := "SrcType := Int" } EQ_Contact(in1 := #Conv_Pos_PV, in2 := 7)
   END_RUNG wire#w22
   RUNG wire#w1
      Contact( #iAuto )
      wire#w23
      { S7_Templates := "SrcType := Int" } EQ_Contact(in1 := #iAListNumber, in2 := 8)
      wire#w24
      I_Contact( #iIndexTableON )
      wire#w25
      Coil( #oPosOK[8] )
   END_RUNG
   RUNG wire#w1
      Contact( #iManual )
   END_RUNG wire#w23
   RUNG wire#w1
      Contact( #iManual )
      { S7_Templates := "SrcType := Int" } EQ_Contact(in1 := #iMListNumber, in2 := 8)
   END_RUNG wire#w24
   RUNG wire#w24
      Contact( #iIndexTableON )
      { S7_Templates := "SrcType := Int" } EQ_Contact(in1 := #Conv_Pos_PV, in2 := 8)
   END_RUNG wire#w25
   RUNG wire#w1
      Contact( #iAuto )
      wire#w26
      { S7_Templates := "SrcType := Int" } EQ_Contact(in1 := #iAListNumber, in2 := 9)
      wire#w27
      I_Contact( #iIndexTableON )
      wire#w28
      Coil( #oPosOK[9] )
   END_RUNG
   RUNG wire#w1
      Contact( #iManual )
   END_RUNG wire#w26
   RUNG wire#w1
      Contact( #iManual )
      { S7_Templates := "SrcType := Int" } EQ_Contact(in1 := #iMListNumber, in2 := 9)
   END_RUNG wire#w27
   RUNG wire#w27
      Contact( #iIndexTableON )
      { S7_Templates := "SrcType := Int" } EQ_Contact(in1 := #Conv_Pos_PV, in2 := 9)
   END_RUNG wire#w28
   RUNG wire#w1
      Contact( #iAuto )
      wire#w29
      { S7_Templates := "SrcType := Int" } EQ_Contact(in1 := #iAListNumber, in2 := 10)
      wire#w30
      I_Contact( #iIndexTableON )
      wire#w31
      Coil( #oPosOK[10] )
   END_RUNG
   RUNG wire#w1
      Contact( #iManual )
   END_RUNG wire#w29
   RUNG wire#w1
      Contact( #iManual )
      { S7_Templates := "SrcType := Int" } EQ_Contact(in1 := #iMListNumber, in2 := 10)
   END_RUNG wire#w30
   RUNG wire#w30
      Contact( #iIndexTableON )
      { S7_Templates := "SrcType := Int" } EQ_Contact(in1 := #Conv_Pos_PV, in2 := 10)
   END_RUNG wire#w31
   // the same network as SCL:
   #_w1 := #tNormalON AND #sCMMT.AxisPosOk AND #sPosOK AND NOT #sRunning;
   #oPosOK[1] := #_w1 AND (((#iAuto OR #iManual) AND (#iAListNumber = 1)) OR (#iManual AND (#iMListNumber = 1))) AND (NOT #iIndexTableON OR (#iIndexTableON AND (#Conv_Pos_PV = 1)));
   #oPosOK[2] := #_w1 AND (((#iAuto OR #iManual) AND (#iAListNumber = 2)) OR (#iManual AND (#iMListNumber = 2))) AND (NOT #iIndexTableON OR (#iIndexTableON AND (#Conv_Pos_PV = 2)));
   #oPosOK[3] := #_w1 AND (((#iAuto OR #iManual) AND (#iAListNumber = 3)) OR (#iManual AND (#iMListNumber = 3))) AND (NOT #iIndexTableON OR (#iIndexTableON AND (#Conv_Pos_PV = 3)));
   #oPosOK[4] := #_w1 AND (((#iAuto OR #iManual) AND (#iAListNumber = 4)) OR (#iManual AND (#iMListNumber = 4))) AND (NOT #iIndexTableON OR (#iIndexTableON AND (#Conv_Pos_PV = 4)));
   #oPosOK[5] := #_w1 AND (((#iAuto OR #iManual) AND (#iAListNumber = 5)) OR (#iManual AND (#iMListNumber = 5))) AND (NOT #iIndexTableON OR (#iIndexTableON AND (#Conv_Pos_PV = 5)));
   #oPosOK[6] := #_w1 AND (((#iAuto OR #iManual) AND (#iAListNumber = 6)) OR (#iManual AND (#iMListNumber = 6))) AND (NOT #iIndexTableON OR (#iIndexTableON AND (#Conv_Pos_PV = 6)));
   #oPosOK[7] := #_w1 AND (((#iAuto OR #iManual) AND (#iAListNumber = 7)) OR (#iManual AND (#iMListNumber = 7))) AND (NOT #iIndexTableON OR (#iIndexTableON AND (#Conv_Pos_PV = 7)));
   #oPosOK[8] := #_w1 AND (((#iAuto OR #iManual) AND (#iAListNumber = 8)) OR (#iManual AND (#iMListNumber = 8))) AND (NOT #iIndexTableON OR (#iIndexTableON AND (#Conv_Pos_PV = 8)));
   #oPosOK[9] := #_w1 AND (((#iAuto OR #iManual) AND (#iAListNumber = 9)) OR (#iManual AND (#iMListNumber = 9))) AND (NOT #iIndexTableON OR (#iIndexTableON AND (#Conv_Pos_PV = 9)));
   #oPosOK[10] := #_w1 AND (((#iAuto OR #iManual) AND (#iAListNumber = 10)) OR (#iManual AND (#iMListNumber = 10))) AND (NOT #iIndexTableON OR (#iIndexTableON AND (#Conv_Pos_PV = 10)));
END_REGION

REGION Network 20: Output Status
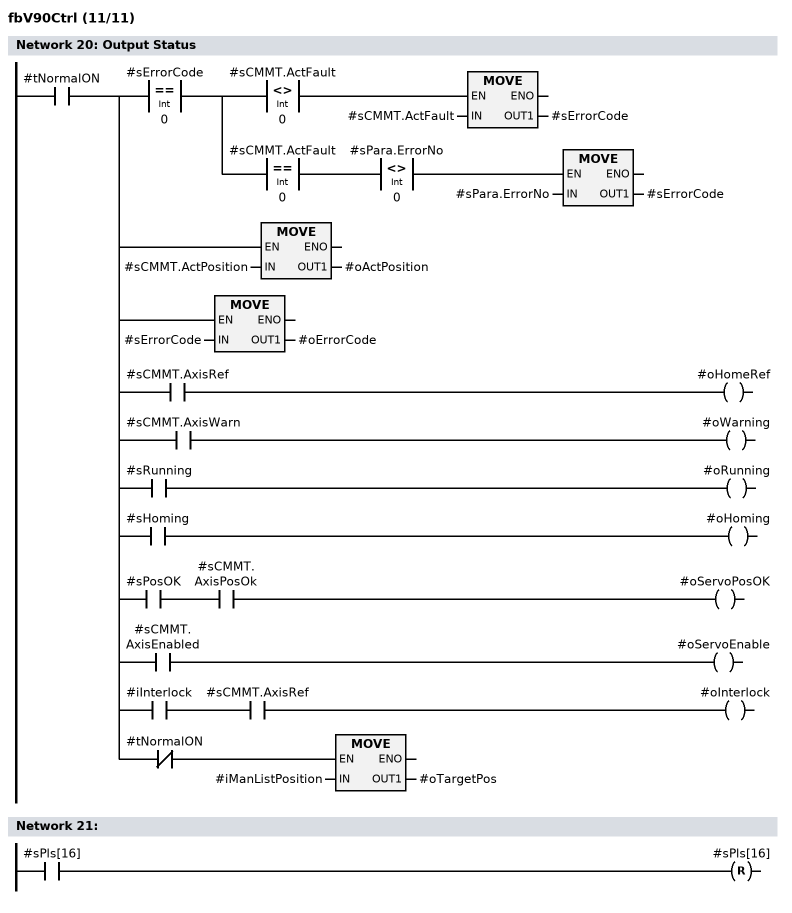
   RUNG wire#powerrail
      Contact( #tNormalON )
      wire#w1
      { S7_Templates := "SrcType := Int" } EQ_Contact(in1 := #sErrorCode, in2 := 0)
      wire#w2
      { S7_Templates := "SrcType := Int" } NE_Contact(in1 := #sCMMT.ActFault, in2 := 0)
      Move(in := #sCMMT.ActFault, out1 => #sErrorCode)
   END_RUNG
   RUNG wire#w2
      { S7_Templates := "SrcType := Int" } EQ_Contact(in1 := #sCMMT.ActFault, in2 := 0)
      { S7_Templates := "SrcType := Int" } NE_Contact(in1 := #sPara.ErrorNo, in2 := 0)
      Move(in := #sPara.ErrorNo, out1 => #sErrorCode)
   END_RUNG
   RUNG wire#w1
      Move(in := #sCMMT.ActPosition, out1 => #oActPosition)
   END_RUNG
   RUNG wire#w1
      Move(in := #sErrorCode, out1 => #oErrorCode)
   END_RUNG
   RUNG wire#w1
      Contact( #sCMMT.AxisRef )
      Coil( #oHomeRef )
   END_RUNG
   RUNG wire#w1
      Contact( #sCMMT.AxisWarn )
      Coil( #oWarning )
   END_RUNG
   RUNG wire#w1
      Contact( #sRunning )
      Coil( #oRunning )
   END_RUNG
   RUNG wire#w1
      Contact( #sHoming )
      Coil( #oHoming )
   END_RUNG
   RUNG wire#w1
      Contact( #sPosOK )
      Contact( #sCMMT.AxisPosOk )
      Coil( #oServoPosOK )
   END_RUNG
   RUNG wire#w1
      Contact( #sCMMT.AxisEnabled )
      Coil( #oServoEnable )
   END_RUNG
   RUNG wire#w1
      Contact( #iInterlock )
      Contact( #sCMMT.AxisRef )
      Coil( #oInterlock )
   END_RUNG
   RUNG wire#w1
      I_Contact( #tNormalON )
      Move(in := #iManListPosition, out1 => #oTargetPos)
   END_RUNG
   // the same network as SCL:
   #_w1 := #tNormalON AND (#sErrorCode = 0);
   IF #_w1 AND (#sCMMT.ActFault <> 0) THEN #sErrorCode := #sCMMT.ActFault; END_IF;
   IF #_w1 AND (#sCMMT.ActFault = 0) AND (#sPara.ErrorNo <> 0) THEN #sErrorCode := #sPara.ErrorNo; END_IF;
   IF #tNormalON THEN
       #oActPosition := #sCMMT.ActPosition;
       #oErrorCode := #sErrorCode;
   END_IF;
   #oHomeRef := #tNormalON AND #sCMMT.AxisRef;
   #oWarning := #tNormalON AND #sCMMT.AxisWarn;
   #oRunning := #tNormalON AND #sRunning;
   #oHoming := #tNormalON AND #sHoming;
   #oServoPosOK := #tNormalON AND #sPosOK AND #sCMMT.AxisPosOk;
   #oServoEnable := #tNormalON AND #sCMMT.AxisEnabled;
   #oInterlock := #tNormalON AND #iInterlock AND #sCMMT.AxisRef;
   IF #tNormalON AND NOT #tNormalON THEN #oTargetPos := #iManListPosition; END_IF;
END_REGION

REGION Network 21
   RUNG wire#powerrail
      Contact( #sPls[16] )
      R_Coil( #sPls[16] )
   END_RUNG
   // the same network as SCL:
   IF #sPls[16] THEN #sPls[16] := FALSE; END_IF;
END_REGION
END_FUNCTION_BLOCK

